LIN {X 0,Y 229.411,Z 367.195,A -85,B 0,C 180,E1 -21102.467,E2 -21102.467} C_VEL
LIN {X 0,Y 228.423,Z 377.715,A -85,B 0,C 180,E1 -21103.053,E2 -21103.053} C_VEL
LIN {X 0,Y 226.714,Z 389.278,A -85,B 0,C 180,E1 -21104.045,E2 -21104.045} C_VEL
LIN {X 0,Y 225.078,Z 397.764,A -85,B 0,C 180,E1 -21105.053,E2 -21105.053} C_VEL
LIN {X 0,Y 223.008,Z 406.34,A -85,B 0,C 180,E1 -21106.348,E2 -21106.348} C_VEL
LIN {X 0,Y 221.124,Z 413.107,A -85,B 0,C 180,E1 -21107.61,E2 -21107.61} C_VEL
LIN {X 0,Y 218.634,Z 420.799,A -85,B 0,C 180,E1 -21109.388,E2 -21109.388} C_VEL
LIN {X 0,Y 216.972,Z 425.412,A -85,B 0,C 180,E1 -21110.663,E2 -21110.663} C_VEL
LIN {X 0,Y 214.589,Z 431.432,A -85,B 0,C 180,E1 -21112.707,E2 -21112.707} C_VEL
LIN {X 0,Y 212.554,Z 436.048,A -85,B 0,C 180,E1 -21114.646,E2 -21114.646} C_VEL
LIN {X 0,Y 210.526,Z 440.403,A -85,B 0,C 180,E1 -21116.988,E2 -21116.988} C_VEL
LIN {X 0,Y 208.603,Z 444.082,A -85,B 0,C 180,E1 -21119.645,E2 -21119.645} C_VEL
LIN {X 0,Y 207.361,Z 446.196,A -85,B 0,C 180,E1 -21121.771,E2 -21121.771} C_VEL
LIN {X 0,Y 206.384,Z 447.588,A -85,B 0,C 180,E1 -21123.725,E2 -21123.725} C_VEL
LIN {X 0,Y 205.598,Z 448.503,A -85,B 0,C 180,E1 -21125.783,E2 -21125.783} C_VEL
LIN {X 0,Y 205.017,Z 448.806,A -85,B 0,C 180,E1 -21127.847,E2 -21127.847} C_VEL
LIN {X 0,Y 204.612,Z 448.539,A -85,B 0,C 180,E1 -21129.911,E2 -21129.911} C_VEL
LIN {X 0,Y 204.369,Z 447.762,A -85,B 0,C 180,E1 -21131.971,E2 -21131.971} C_VEL
LIN {X 0,Y 204.347,Z 446.209,A -85,B 0,C 180,E1 -21134.332,E2 -21134.332} C_VEL
LIN {X 0,Y 204.576,Z 443.416,A -85,B 0,C 180,E1 -21137.097,E2 -21137.097} C_VEL
LIN {X 0,Y 204.907,Z 440.635,A -85,B 0,C 180,E1 -21139.127,E2 -21139.127} C_VEL
LIN {X 0,Y 205.336,Z 437.209,A -85,B 0,C 180,E1 -21141.14,E2 -21141.14} C_VEL
LIN {X 0,Y 205.954,Z 432.897,A -85,B 0,C 180,E1 -21143.201,E2 -21143.201} C_VEL
LIN {X 0,Y 206.566,Z 428.044,A -85,B 0,C 180,E1 -21145.121,E2 -21145.121} C_VEL
LIN {X 0,Y 207.459,Z 421.98,A -85,B 0,C 180,E1 -21147.088,E2 -21147.088} C_VEL
LIN {X 0,Y 208.512,Z 414.595,A -85,B 0,C 180,E1 -21149.035,E2 -21149.035} C_VEL
LIN {X 0,Y 209.626,Z 406.687,A -85,B 0,C 180,E1 -21150.721,E2 -21150.721} C_VEL
LIN {X 0,Y 210.63,Z 398.846,A -85,B 0,C 180,E1 -21152.072,E2 -21152.072} C_VEL
LIN {X 0,Y 211.564,Z 389.853,A -85,B 0,C 180,E1 -21153.307,E2 -21153.307} C_VEL
LIN {X 0,Y 212.44,Z 379.124,A -85,B 0,C 180,E1 -21154.418,E2 -21154.418} C_VEL
LIN {X 0,Y 213.039,Z 367.681,A -85,B 0,C 180,E1 -21155.183,E2 -21155.183} C_VEL
LIN {X 0,Y 213.743,Z 344.69,A -85,B 0,C 180,E1 -21156.017,E2 -21156.017} C_VEL
LIN {X 0,Y 214.449,Z 316.245,A -85,B 0,C 180,E1 -21156.958,E2 -21156.958} C_VEL
LIN {X 0,Y 213.406,Z 311.932,A -85,B 0,C 180,E1 -21157.204,E2 -21157.204} C_VEL
LIN {X 0,Y 207.738,Z 296.649,A -85,B 0,C 180,E1 -21158.29,E2 -21158.29} C_VEL
LIN {X 0,Y 207.116,Z 294.495,A -85,B 0,C 180,E1 -21158.446,E2 -21158.446} C_VEL
LIN {X 0,Y 206.854,Z 294.531,A -85,B 0,C 180,E1 -21163.759,E2 -21163.759} C_VEL
LIN {X 0,Y 206.829,Z 294.533,A -85,B 0,C 180,E1 -21167.957,E2 -21167.957} C_VEL
LIN {X 0,Y 206.719,Z 294.549,A -85,B 0,C 180,E1 -21173.394,E2 -21173.394} C_VEL
LIN {X 0,Y 206.663,Z 294.553,A -85,B 0,C 180,E1 -21178.431,E2 -21178.431} C_VEL
LIN {X 0,Y 206.67,Z 294.546,A -85,B 0,C 180,E1 -21182.963,E2 -21182.963} C_VEL
LIN {X 0,Y 206.646,Z 294.553,A -85,B 0,C 180,E1 -21187.748,E2 -21187.748} C_VEL
LIN {X 0,Y 206.614,Z 294.561,A -85,B 0,C 180,E1 -21191.566,E2 -21191.566} C_VEL
LIN {X 0,Y 206.612,Z 294.559,A -85,B 0,C 180,E1 -21195.588,E2 -21195.588} C_VEL
LIN {X 0,Y 206.643,Z 294.555,A -85,B 0,C 180,E1 -21199.755,E2 -21199.755} C_VEL
LIN {X 0,Y 206.685,Z 294.55,A -85,B 0,C 180,E1 -21204.695,E2 -21204.695} C_VEL
LIN {X 0,Y 206.684,Z 294.549,A -85,B 0,C 180,E1 -21209.341,E2 -21209.341} C_VEL
LIN {X 0,Y 206.696,Z 294.55,A -85,B 0,C 180,E1 -21213.775,E2 -21213.775} C_VEL
LIN {X 0,Y 206.742,Z 294.526,A -85,B 0,C 180,E1 -21218.049,E2 -21218.049} C_VEL
LIN {X 0,Y 207.124,Z 294.503,A -85,B 0,C 180,E1 -21222.354,E2 -21222.354} C_VEL
LIN {X 0,Y 208.929,Z 312.159,A -85,B 0,C 180,E1 -21223.393,E2 -21223.393} C_VEL
LIN {X 0,Y 207.623,Z 366.937,A -85,B 0,C 180,E1 -21226.799,E2 -21226.799} C_VEL
LIN {X 0,Y 207.292,Z 379.206,A -85,B 0,C 180,E1 -21227.897,E2 -21227.897} C_VEL
LIN {X 0,Y 206.834,Z 390.233,A -85,B 0,C 180,E1 -21229.236,E2 -21229.236} C_VEL
LIN {X 0,Y 206.324,Z 400.757,A -85,B 0,C 180,E1 -21230.942,E2 -21230.942} C_VEL
LIN {X 0,Y 205.886,Z 409.682,A -85,B 0,C 180,E1 -21232.727,E2 -21232.727} C_VEL
LIN {X 0,Y 205.418,Z 419.232,A -85,B 0,C 180,E1 -21235.1,E2 -21235.1} C_VEL
LIN {X 0,Y 205.266,Z 425.662,A -85,B 0,C 180,E1 -21237.063,E2 -21237.063} C_VEL
LIN {X 0,Y 204.925,Z 432.222,A -85,B 0,C 180,E1 -21239.515,E2 -21239.515} C_VEL
LIN {X 0,Y 204.912,Z 437.509,A -85,B 0,C 180,E1 -21241.972,E2 -21241.972} C_VEL
LIN {X 0,Y 205.35,Z 442.572,A -85,B 0,C 180,E1 -21244.914,E2 -21244.914} C_VEL
LIN {X 0,Y 206.174,Z 446.28,A -85,B 0,C 180,E1 -21247.843,E2 -21247.843} C_VEL
LIN {X 0,Y 207.385,Z 448.706,A -85,B 0,C 180,E1 -21250.649,E2 -21250.649} C_VEL
LIN {X 0,Y 209.615,Z 450.18,A -85,B 0,C 180,E1 -21253.58,E2 -21253.58} C_VEL
LIN {X 0,Y 211.19,Z 450.591,A -85,B 0,C 180,E1 -21255.445,E2 -21255.445} C_VEL
LIN {X 0,Y 213.288,Z 450.479,A -85,B 0,C 180,E1 -21257.257,E2 -21257.257} C_VEL
LIN {X 0,Y 215.528,Z 449.821,A -85,B 0,C 180,E1 -21259.037,E2 -21259.037} C_VEL
LIN {X 0,Y 217.99,Z 448.714,A -85,B 0,C 180,E1 -21260.777,E2 -21260.777} C_VEL
LIN {X 0,Y 222.26,Z 446.105,A -85,B 0,C 180,E1 -21263.288,E2 -21263.288} C_VEL
LIN {X 0,Y 226.988,Z 442.34,A -85,B 0,C 180,E1 -21265.693,E2 -21265.693} C_VEL
LIN {X 0,Y 232.158,Z 437.117,A -85,B 0,C 180,E1 -21267.989,E2 -21267.989} C_VEL
LIN {X 0,Y 236.824,Z 431.622,A -85,B 0,C 180,E1 -21269.812,E2 -21269.812} C_VEL
LIN {X 0,Y 241.781,Z 424.82,A -85,B 0,C 180,E1 -21271.553,E2 -21271.553} C_VEL
LIN {X 0,Y 247.029,Z 416.545,A -85,B 0,C 180,E1 -21273.212,E2 -21273.212} C_VEL
LIN {X 0,Y 251.926,Z 407.174,A -85,B 0,C 180,E1 -21274.644,E2 -21274.644} C_VEL
LIN {X 0,Y 253.424,Z 404.07,A -85,B 0,C 180,E1 -21275.039,E2 -21275.039} C_VEL
LIN {X 0,Y 254.666,Z 401.027,A -85,B 0,C 180,E1 -21275.561,E2 -21275.561} C_VEL
LIN {X 0,Y 256.581,Z 392.474,A -85,B 0,C 180,E1 -21277.676,E2 -21277.676} C_VEL
LIN {X 0,Y 257.472,Z 389.198,A -85,B 0,C 180,E1 -21278.133,E2 -21278.133} C_VEL
LIN {X 0,Y 257.664,Z 388.604,A -85,B 0,C 180,E1 -21278.182,E2 -21278.182} C_VEL
LIN {X 0,Y 260.972,Z 377.957,A -85,B 0,C 180,E1 -21278.916,E2 -21278.916} C_VEL
LIN {X 0,Y 262.394,Z 372.569,A -85,B 0,C 180,E1 -21279.217,E2 -21279.217} C_VEL
LIN {X 0,Y 261.762,Z 370.849,A -85,B 0,C 180,E1 -21280.53,E2 -21280.53} C_VEL
LIN {X 0,Y 261.245,Z 369.295,A -85,B 0,C 180,E1 -21282.269,E2 -21282.269} C_VEL
LIN {X 0,Y 260.914,Z 369.054,A -85,B 0,C 180,E1 -21285.545,E2 -21285.545} C_VEL
LIN {X 0,Y 261.153,Z 369.578,A -85,B 0,C 180,E1 -21287,E2 -21287} C_VEL
LIN {X 0,Y 262.17,Z 372.974,A -85,B 0,C 180,E1 -21289.887,E2 -21289.887} C_VEL
LIN {X 0,Y 262.361,Z 373.577,A -85,B 0,C 180,E1 -21290.252,E2 -21290.252} C_VEL
LIN {X 0,Y 258.592,Z 387.877,A -85,B 0,C 180,E1 -21291.027,E2 -21291.027} C_VEL
LIN {X 0,Y 254.187,Z 400.181,A -85,B 0,C 180,E1 -21291.85,E2 -21291.85} C_VEL
LIN {X 0,Y 248.945,Z 411.733,A -85,B 0,C 180,E1 -21292.883,E2 -21292.883} C_VEL
LIN {X 0,Y 243.475,Z 421.754,A -85,B 0,C 180,E1 -21294.087,E2 -21294.087} C_VEL
LIN {X 0,Y 237.019,Z 431.728,A -85,B 0,C 180,E1 -21295.71,E2 -21295.71} C_VEL
LIN {X 0,Y 231.35,Z 439.3,A -85,B 0,C 180,E1 -21297.369,E2 -21297.369} C_VEL
LIN {X 0,Y 225.07,Z 446.659,A -85,B 0,C 180,E1 -21299.507,E2 -21299.507} C_VEL
LIN {X 0,Y 220.232,Z 451.53,A -85,B 0,C 180,E1 -21301.4,E2 -21301.4} C_VEL
LIN {X 0,Y 215.03,Z 456.023,A -85,B 0,C 180,E1 -21303.817,E2 -21303.817} C_VEL
LIN {X 0,Y 210.452,Z 459.369,A -85,B 0,C 180,E1 -21306.375,E2 -21306.375} C_VEL
LIN {X 0,Y 207.759,Z 461.023,A -85,B 0,C 180,E1 -21308.154,E2 -21308.154} C_VEL
LIN {X 0,Y 205.278,Z 462.198,A -85,B 0,C 180,E1 -21309.979,E2 -21309.979} C_VEL
LIN {X 0,Y 203.302,Z 462.83,A -85,B 0,C 180,E1 -21311.873,E2 -21311.873} C_VEL
LIN {X 0,Y 200.363,Z 462.941,A -85,B 0,C 180,E1 -21315.786,E2 -21315.786} C_VEL
LIN {X 0,Y 199.313,Z 462.261,A -85,B 0,C 180,E1 -21317.785,E2 -21317.785} C_VEL
LIN {X 0,Y 198.285,Z 459.599,A -85,B 0,C 180,E1 -21321.849,E2 -21321.849} C_VEL
LIN {X 0,Y 198.2,Z 458.32,A -85,B 0,C 180,E1 -21323.293,E2 -21323.293} C_VEL
LIN {X 0,Y 197.665,Z 461.871,A -85,B 0,C 180,E1 -21325.922,E2 -21325.922} C_VEL
LIN {X 0,Y 197.59,Z 463.98,A -85,B 0,C 180,E1 -21327.961,E2 -21327.961} C_VEL
LIN {X 0,Y 197.617,Z 465.545,A -85,B 0,C 180,E1 -21330,E2 -21330} C_VEL
LIN {X 0,Y 197.498,Z 466.482,A -85,B 0,C 180,E1 -21332.039,E2 -21332.039} C_VEL
LIN {X 0,Y 197.419,Z 466.975,A -85,B 0,C 180,E1 -21334.542,E2 -21334.542} C_VEL
LIN {X 0,Y 197.725,Z 466.437,A -85,B 0,C 180,E1 -21338.173,E2 -21338.173} C_VEL
LIN {X 0,Y 198.227,Z 465.424,A -85,B 0,C 180,E1 -21340.21,E2 -21340.21} C_VEL
LIN {X 0,Y 199.459,Z 462.979,A -85,B 0,C 180,E1 -21343.24,E2 -21343.24} C_VEL
LIN {X 0,Y 201.207,Z 459.238,A -85,B 0,C 180,E1 -21346.226,E2 -21346.226} C_VEL
LIN {X 0,Y 202.731,Z 456.069,A -85,B 0,C 180,E1 -21348.179,E2 -21348.179} C_VEL
LIN {X 0,Y 205.071,Z 451.053,A -85,B 0,C 180,E1 -21350.565,E2 -21350.565} C_VEL
LIN {X 0,Y 207.767,Z 444.774,A -85,B 0,C 180,E1 -21352.892,E2 -21352.892} C_VEL
LIN {X 0,Y 210.188,Z 438.652,A -85,B 0,C 180,E1 -21354.705,E2 -21354.705} C_VEL
LIN {X 0,Y 212.071,Z 433.271,A -85,B 0,C 180,E1 -21356.046,E2 -21356.046} C_VEL
LIN {X 0,Y 214.178,Z 426.968,A -85,B 0,C 180,E1 -21357.348,E2 -21357.348} C_VEL
LIN {X 0,Y 216.962,Z 417.427,A -85,B 0,C 180,E1 -21358.886,E2 -21358.886} C_VEL
LIN {X 0,Y 218.812,Z 409.826,A -85,B 0,C 180,E1 -21359.856,E2 -21359.856} C_VEL
LIN {X 0,Y 220.554,Z 401.702,A -85,B 0,C 180,E1 -21360.653,E2 -21360.653} C_VEL
LIN {X 0,Y 222.104,Z 392.178,A -85,B 0,C 180,E1 -21361.346,E2 -21361.346} C_VEL
LIN {X 0,Y 223.067,Z 382.979,A -85,B 0,C 180,E1 -21361.814,E2 -21361.814} C_VEL
LIN {X 0,Y 224.088,Z 362.598,A -85,B 0,C 180,E1 -21362.502,E2 -21362.502} C_VEL
LIN {X 0,Y 221.37,Z 343.446,A -85,B 0,C 180,E1 -21363.879,E2 -21363.879} C_VEL
LIN {X 0,Y 220.472,Z 339.745,A -85,B 0,C 180,E1 -21364.235,E2 -21364.235} C_VEL
LIN {X 0,Y 215.073,Z 327.747,A -85,B 0,C 180,E1 -21366.016,E2 -21366.016} C_VEL
LIN {X 0,Y 209.948,Z 317.918,A -85,B 0,C 180,E1 -21367.766,E2 -21367.766} C_VEL
LIN {X 0,Y 207.328,Z 313.245,A -85,B 0,C 180,E1 -21368.696,E2 -21368.696} C_VEL
LIN {X 0,Y 204.763,Z 308.846,A -85,B 0,C 180,E1 -21369.638,E2 -21369.638} C_VEL
LIN {X 0,Y 202.164,Z 304.496,A -85,B 0,C 180,E1 -21370.632,E2 -21370.632} C_VEL
LIN {X 0,Y 201.935,Z 303.874,A -85,B 0,C 180,E1 -21370.819,E2 -21370.819} C_VEL
LIN {X 0,Y 200.406,Z 298.59,A -85,B 0,C 180,E1 -21374.537,E2 -21374.537} C_VEL
LIN {X 0,Y 199.607,Z 295.427,A -85,B 0,C 180,E1 -21377.05,E2 -21377.05} C_VEL
LIN {X 0,Y 199.606,Z 295.424,A -85,B 0,C 180,E1 -21380.769,E2 -21380.769} C_VEL
LIN {X 0,Y 199.619,Z 295.423,A -85,B 0,C 180,E1 -21385.708,E2 -21385.708} C_VEL
LIN {X 0,Y 199.694,Z 295.414,A -85,B 0,C 180,E1 -21388.13,E2 -21388.13} C_VEL
LIN {X 0,Y 199.651,Z 295.419,A -85,B 0,C 180,E1 -21392.76,E2 -21392.76} C_VEL
LIN {X 0,Y 199.715,Z 295.413,A -85,B 0,C 180,E1 -21397.22,E2 -21397.22} C_VEL
LIN {X 0,Y 199.801,Z 295.405,A -85,B 0,C 180,E1 -21401.754,E2 -21401.754} C_VEL
LIN {X 0,Y 199.828,Z 295.4,A -85,B 0,C 180,E1 -21405.742,E2 -21405.742} C_VEL
LIN {X 0,Y 200.026,Z 295.362,A -85,B 0,C 180,E1 -21409.876,E2 -21409.876} C_VEL
LIN {X 0,Y 200.02,Z 295.362,A -85,B 0,C 180,E1 -21413.943,E2 -21413.943} C_VEL
LIN {X 0,Y 200.316,Z 295.336,A -85,B 0,C 180,E1 -21417.983,E2 -21417.983} C_VEL
LIN {X 0,Y 200.473,Z 295.305,A -85,B 0,C 180,E1 -21419.994,E2 -21419.994} C_VEL
LIN {X 0,Y 200.016,Z 295.37,A -85,B 0,C 180,E1 -21424.023,E2 -21424.023} C_VEL
LIN {X 0,Y 200.079,Z 295.374,A -85,B 0,C 180,E1 -21428.07,E2 -21428.07} C_VEL
LIN {X 0,Y 199.87,Z 295.395,A -85,B 0,C 180,E1 -21432.173,E2 -21432.173} C_VEL
LIN {X 0,Y 199.797,Z 295.398,A -85,B 0,C 180,E1 -21436.337,E2 -21436.337} C_VEL
LIN {X 0,Y 199.694,Z 295.411,A -85,B 0,C 180,E1 -21440.598,E2 -21440.598} C_VEL
LIN {X 0,Y 199.662,Z 295.418,A -85,B 0,C 180,E1 -21444.978,E2 -21444.978} C_VEL
LIN {X 0,Y 199.651,Z 295.425,A -85,B 0,C 180,E1 -21449.517,E2 -21449.517} C_VEL
LIN {X 0,Y 199.677,Z 295.469,A -85,B 0,C 180,E1 -21451.784,E2 -21451.784} C_VEL
LIN {X 0,Y 200.481,Z 297.963,A -85,B 0,C 180,E1 -21452.178,E2 -21452.178} C_VEL
LIN {X 0,Y 202.382,Z 300.199,A -85,B 0,C 180,E1 -21452.885,E2 -21452.885} C_VEL
LIN {X 0,Y 203.114,Z 301.083,A -85,B 0,C 180,E1 -21453.153,E2 -21453.153} C_VEL
LIN {X 0,Y 205.286,Z 304.358,A -85,B 0,C 180,E1 -21453.958,E2 -21453.958} C_VEL
LIN {X 0,Y 210.304,Z 311.674,A -85,B 0,C 180,E1 -21455.703,E2 -21455.703} C_VEL
LIN {X 0,Y 216.59,Z 321.533,A -85,B 0,C 180,E1 -21457.743,E2 -21457.743} C_VEL
LIN {X 0,Y 222.99,Z 333.019,A -85,B 0,C 180,E1 -21459.703,E2 -21459.703} C_VEL
LIN {X 0,Y 225.333,Z 338.511,A -85,B 0,C 180,E1 -21460.432,E2 -21460.432} C_VEL
LIN {X 0,Y 223.827,Z 366.884,A -85,B 0,C 180,E1 -21461.355,E2 -21461.355} C_VEL
LIN {X 0,Y 222.95,Z 376.004,A -85,B 0,C 180,E1 -21461.841,E2 -21461.841} C_VEL
LIN {X 0,Y 221.602,Z 385.861,A -85,B 0,C 180,E1 -21462.623,E2 -21462.623} C_VEL
LIN {X 0,Y 219.46,Z 397.28,A -85,B 0,C 180,E1 -21463.901,E2 -21463.901} C_VEL
LIN {X 0,Y 217.173,Z 406.269,A -85,B 0,C 180,E1 -21465.259,E2 -21465.259} C_VEL
LIN {X 0,Y 214.687,Z 414.699,A -85,B 0,C 180,E1 -21466.893,E2 -21466.893} C_VEL
LIN {X 0,Y 212.346,Z 421.559,A -85,B 0,C 180,E1 -21468.552,E2 -21468.552} C_VEL
LIN {X 0,Y 209.84,Z 428.001,A -85,B 0,C 180,E1 -21470.48,E2 -21470.48} C_VEL
LIN {X 0,Y 206.985,Z 434.507,A -85,B 0,C 180,E1 -21472.938,E2 -21472.938} C_VEL
LIN {X 0,Y 204.46,Z 439.725,A -85,B 0,C 180,E1 -21475.571,E2 -21475.571} C_VEL
LIN {X 0,Y 202.141,Z 443.96,A -85,B 0,C 180,E1 -21478.566,E2 -21478.566} C_VEL
LIN {X 0,Y 200.544,Z 446.53,A -85,B 0,C 180,E1 -21481.16,E2 -21481.16} C_VEL
LIN {X 0,Y 199.69,Z 447.732,A -85,B 0,C 180,E1 -21482.773,E2 -21482.773} C_VEL
LIN {X 0,Y 198.808,Z 448.703,A -85,B 0,C 180,E1 -21484.9,E2 -21484.9} C_VEL
LIN {X 0,Y 198.061,Z 449.116,A -85,B 0,C 180,E1 -21487.285,E2 -21487.285} C_VEL
LIN {X 0,Y 197.642,Z 448.943,A -85,B 0,C 180,E1 -21489.171,E2 -21489.171} C_VEL
LIN {X 0,Y 197.328,Z 448.293,A -85,B 0,C 180,E1 -21491.305,E2 -21491.305} C_VEL
LIN {X 0,Y 197.254,Z 446.572,A -85,B 0,C 180,E1 -21494.12,E2 -21494.12} C_VEL
LIN {X 0,Y 197.411,Z 444.21,A -85,B 0,C 180,E1 -21496.621,E2 -21496.621} C_VEL
LIN {X 0,Y 197.924,Z 439.995,A -85,B 0,C 180,E1 -21499.774,E2 -21499.774} C_VEL
LIN {X 0,Y 198.554,Z 435.513,A -85,B 0,C 180,E1 -21502.28,E2 -21502.28} C_VEL
LIN {X 0,Y 199.396,Z 429.454,A -85,B 0,C 180,E1 -21504.945,E2 -21504.945} C_VEL
LIN {X 0,Y 200.517,Z 421.898,A -85,B 0,C 180,E1 -21507.489,E2 -21507.489} C_VEL
LIN {X 0,Y 201.603,Z 414.437,A -85,B 0,C 180,E1 -21509.501,E2 -21509.501} C_VEL
LIN {X 0,Y 202.77,Z 406.431,A -85,B 0,C 180,E1 -21511.242,E2 -21511.242} C_VEL
LIN {X 0,Y 204.042,Z 396.843,A -85,B 0,C 180,E1 -21512.894,E2 -21512.894} C_VEL
LIN {X 0,Y 205.137,Z 385.908,A -85,B 0,C 180,E1 -21514.298,E2 -21514.298} C_VEL
LIN {X 0,Y 205.853,Z 376.021,A -85,B 0,C 180,E1 -21515.204,E2 -21515.204} C_VEL
LIN {X 0,Y 206.3,Z 366.415,A -85,B 0,C 180,E1 -21515.805,E2 -21515.805} C_VEL
LIN {X 0,Y 207.728,Z 317.216,A -85,B 0,C 180,E1 -21517.537,E2 -21517.537} C_VEL
LIN {X 0,Y 206.282,Z 312.34,A -85,B 0,C 180,E1 -21517.854,E2 -21517.854} C_VEL
LIN {X 0,Y 200.994,Z 298.072,A -85,B 0,C 180,E1 -21518.919,E2 -21518.919} C_VEL
LIN {X 0,Y 200.042,Z 295.378,A -85,B 0,C 180,E1 -21519.162,E2 -21519.162} C_VEL
LIN {X 0,Y 199.795,Z 295.41,A -85,B 0,C 180,E1 -21524.255,E2 -21524.255} C_VEL
LIN {X 0,Y 199.754,Z 295.414,A -85,B 0,C 180,E1 -21528.461,E2 -21528.461} C_VEL
LIN {X 0,Y 199.681,Z 295.426,A -85,B 0,C 180,E1 -21533.801,E2 -21533.801} C_VEL
LIN {X 0,Y 199.64,Z 295.428,A -85,B 0,C 180,E1 -21538.365,E2 -21538.365} C_VEL
LIN {X 0,Y 199.641,Z 295.42,A -85,B 0,C 180,E1 -21542.357,E2 -21542.357} C_VEL
LIN {X 0,Y 199.595,Z 295.432,A -85,B 0,C 180,E1 -21546.77,E2 -21546.77} C_VEL
LIN {X 0,Y 199.574,Z 295.433,A -85,B 0,C 180,E1 -21549.337,E2 -21549.337} C_VEL
LIN {X 0,Y 199.548,Z 295.438,A -85,B 0,C 180,E1 -21552.314,E2 -21552.314} C_VEL
LIN {X 0,Y 199.558,Z 295.436,A -85,B 0,C 180,E1 -21555.234,E2 -21555.234} C_VEL
LIN {X 0,Y 199.561,Z 295.439,A -85,B 0,C 180,E1 -21558.011,E2 -21558.011} C_VEL
LIN {X 0,Y 199.594,Z 295.429,A -85,B 0,C 180,E1 -21560.774,E2 -21560.774} C_VEL
LIN {X 0,Y 199.598,Z 295.435,A -85,B 0,C 180,E1 -21565.72,E2 -21565.72} C_VEL
LIN {X 0,Y 199.673,Z 295.422,A -85,B 0,C 180,E1 -21568.141,E2 -21568.141} C_VEL
LIN {X 0,Y 199.633,Z 295.428,A -85,B 0,C 180,E1 -21572.772,E2 -21572.772} C_VEL
LIN {X 0,Y 199.706,Z 295.407,A -85,B 0,C 180,E1 -21577.233,E2 -21577.233} C_VEL
LIN {X 0,Y 200.111,Z 295.348,A -85,B 0,C 180,E1 -21582.474,E2 -21582.474} C_VEL
LIN {X 0,Y 201.834,Z 312.319,A -85,B 0,C 180,E1 -21583.508,E2 -21583.508} C_VEL
LIN {X 0,Y 200.597,Z 367.18,A -85,B 0,C 180,E1 -21587.101,E2 -21587.101} C_VEL
LIN {X 0,Y 200.255,Z 379.24,A -85,B 0,C 180,E1 -21588.237,E2 -21588.237} C_VEL
LIN {X 0,Y 199.831,Z 390.259,A -85,B 0,C 180,E1 -21589.623,E2 -21589.623} C_VEL
LIN {X 0,Y 199.322,Z 400.561,A -85,B 0,C 180,E1 -21591.337,E2 -21591.337} C_VEL
LIN {X 0,Y 198.883,Z 409.612,A -85,B 0,C 180,E1 -21593.196,E2 -21593.196} C_VEL
LIN {X 0,Y 198.46,Z 418.538,A -85,B 0,C 180,E1 -21595.437,E2 -21595.437} C_VEL
LIN {X 0,Y 198.182,Z 426.454,A -85,B 0,C 180,E1 -21597.974,E2 -21597.974} C_VEL
LIN {X 0,Y 197.944,Z 432.845,A -85,B 0,C 180,E1 -21600.515,E2 -21600.515} C_VEL
LIN {X 0,Y 198.036,Z 438.096,A -85,B 0,C 180,E1 -21603.058,E2 -21603.058} C_VEL
LIN {X 0,Y 198.602,Z 443.122,A -85,B 0,C 180,E1 -21606.1,E2 -21606.1} C_VEL
LIN {X 0,Y 199.488,Z 446.591,A -85,B 0,C 180,E1 -21608.97,E2 -21608.97} C_VEL
LIN {X 0,Y 201.08,Z 449.222,A -85,B 0,C 180,E1 -21612.111,E2 -21612.111} C_VEL
LIN {X 0,Y 202.736,Z 450.356,A -85,B 0,C 180,E1 -21614.05,E2 -21614.05} C_VEL
LIN {X 0,Y 204.366,Z 450.922,A -85,B 0,C 180,E1 -21615.975,E2 -21615.975} C_VEL
LIN {X 0,Y 206.556,Z 451.016,A -85,B 0,C 180,E1 -21617.838,E2 -21617.838} C_VEL
LIN {X 0,Y 210.298,Z 450.288,A -85,B 0,C 180,E1 -21620.651,E2 -21620.651} C_VEL
LIN {X 0,Y 214.348,Z 448.578,A -85,B 0,C 180,E1 -21623.175,E2 -21623.175} C_VEL
LIN {X 0,Y 219.13,Z 445.649,A -85,B 0,C 180,E1 -21625.662,E2 -21625.662} C_VEL
LIN {X 0,Y 224.371,Z 441.435,A -85,B 0,C 180,E1 -21628.03,E2 -21628.03} C_VEL
LIN {X 0,Y 230.072,Z 435.822,A -85,B 0,C 180,E1 -21630.272,E2 -21630.272} C_VEL
LIN {X 0,Y 236.198,Z 428.724,A -85,B 0,C 180,E1 -21632.389,E2 -21632.389} C_VEL
LIN {X 0,Y 241.606,Z 421.119,A -85,B 0,C 180,E1 -21634.058,E2 -21634.058} C_VEL
LIN {X 0,Y 247.87,Z 410.793,A -85,B 0,C 180,E1 -21635.793,E2 -21635.793} C_VEL
LIN {X 0,Y 252.598,Z 401.229,A -85,B 0,C 180,E1 -21636.994,E2 -21636.994} C_VEL
LIN {X 0,Y 256.461,Z 391.834,A -85,B 0,C 180,E1 -21637.913,E2 -21637.913} C_VEL
LIN {X 0,Y 257.664,Z 388.604,A -85,B 0,C 180,E1 -21638.182,E2 -21638.182} C_VEL
LIN {X 0,Y 258.662,Z 385.151,A -85,B 0,C 180,E1 -21638.594,E2 -21638.594} C_VEL
LIN {X 0,Y 259.267,Z 382.229,A -85,B 0,C 180,E1 -21639.215,E2 -21639.215} C_VEL
LIN {X 0,Y 259.504,Z 379.196,A -85,B 0,C 180,E1 -21640.245,E2 -21640.245} C_VEL
LIN {X 0,Y 259.415,Z 377.14,A -85,B 0,C 180,E1 -21641.413,E2 -21641.413} C_VEL
LIN {X 0,Y 259.3,Z 376.514,A -85,B 0,C 180,E1 -21642.025,E2 -21642.025} C_VEL
LIN {X 0,Y 259.142,Z 375.939,A -85,B 0,C 180,E1 -21642.924,E2 -21642.924} C_VEL
LIN {X 0,Y 259.164,Z 376.017,A -85,B 0,C 180,E1 -21646.177,E2 -21646.177} C_VEL
LIN {X 0,Y 259.289,Z 376.947,A -85,B 0,C 180,E1 -21647.341,E2 -21647.341} C_VEL
LIN {X 0,Y 259.732,Z 378.763,A -85,B 0,C 180,E1 -21648.975,E2 -21648.975} C_VEL
LIN {X 0,Y 255.364,Z 392.759,A -85,B 0,C 180,E1 -21649.758,E2 -21649.758} C_VEL
LIN {X 0,Y 250.507,Z 404.326,A -85,B 0,C 180,E1 -21650.598,E2 -21650.598} C_VEL
LIN {X 0,Y 245.588,Z 413.986,A -85,B 0,C 180,E1 -21651.506,E2 -21651.506} C_VEL
LIN {X 0,Y 238.777,Z 425.141,A -85,B 0,C 180,E1 -21652.94,E2 -21652.94} C_VEL
LIN {X 0,Y 232.723,Z 433.557,A -85,B 0,C 180,E1 -21654.402,E2 -21654.402} C_VEL
LIN {X 0,Y 225.565,Z 442.07,A -85,B 0,C 180,E1 -21656.424,E2 -21656.424} C_VEL
LIN {X 0,Y 220.142,Z 447.633,A -85,B 0,C 180,E1 -21658.213,E2 -21658.213} C_VEL
LIN {X 0,Y 214.115,Z 452.944,A -85,B 0,C 180,E1 -21660.504,E2 -21660.504} C_VEL
LIN {X 0,Y 208.732,Z 457.02,A -85,B 0,C 180,E1 -21662.964,E2 -21662.964} C_VEL
LIN {X 0,Y 203.987,Z 459.927,A -85,B 0,C 180,E1 -21665.578,E2 -21665.578} C_VEL
LIN {X 0,Y 201.199,Z 461.212,A -85,B 0,C 180,E1 -21667.403,E2 -21667.403} C_VEL
LIN {X 0,Y 198.633,Z 462.088,A -85,B 0,C 180,E1 -21669.278,E2 -21669.278} C_VEL
LIN {X 0,Y 196.563,Z 462.583,A -85,B 0,C 180,E1 -21671.228,E2 -21671.228} C_VEL
LIN {X 0,Y 194.886,Z 462.545,A -85,B 0,C 180,E1 -21673.232,E2 -21673.232} C_VEL
LIN {X 0,Y 192.448,Z 461.243,A -85,B 0,C 180,E1 -21677.343,E2 -21677.343} C_VEL
LIN {X 0,Y 191.732,Z 459.964,A -85,B 0,C 180,E1 -21679.439,E2 -21679.439} C_VEL
LIN {X 0,Y 191.314,Z 457.197,A -85,B 0,C 180,E1 -21682.719,E2 -21682.719} C_VEL
LIN {X 0,Y 190.586,Z 461.295,A -85,B 0,C 180,E1 -21685.77,E2 -21685.77} C_VEL
LIN {X 0,Y 190.511,Z 463.478,A -85,B 0,C 180,E1 -21687.885,E2 -21687.885} C_VEL
LIN {X 0,Y 190.552,Z 465.071,A -85,B 0,C 180,E1 -21690,E2 -21690} C_VEL
LIN {X 0,Y 190.413,Z 466.049,A -85,B 0,C 180,E1 -21692.115,E2 -21692.115} C_VEL
LIN {X 0,Y 190.345,Z 466.58,A -85,B 0,C 180,E1 -21694.449,E2 -21694.449} C_VEL
LIN {X 0,Y 190.394,Z 466.605,A -85,B 0,C 180,E1 -21696.357,E2 -21696.357} C_VEL
LIN {X 0,Y 190.7,Z 466.194,A -85,B 0,C 180,E1 -21698.477,E2 -21698.477} C_VEL
LIN {X 0,Y 191.245,Z 465.199,A -85,B 0,C 180,E1 -21700.587,E2 -21700.587} C_VEL
LIN {X 0,Y 192.045,Z 463.712,A -85,B 0,C 180,E1 -21702.684,E2 -21702.684} C_VEL
LIN {X 0,Y 193.727,Z 460.567,A -85,B 0,C 180,E1 -21705.788,E2 -21705.788} C_VEL
LIN {X 0,Y 196.008,Z 456.134,A -85,B 0,C 180,E1 -21708.826,E2 -21708.826} C_VEL
LIN {X 0,Y 198.951,Z 450.055,A -85,B 0,C 180,E1 -21711.772,E2 -21711.772} C_VEL
LIN {X 0,Y 201.263,Z 445.057,A -85,B 0,C 180,E1 -21713.676,E2 -21713.676} C_VEL
LIN {X 0,Y 203.788,Z 439.064,A -85,B 0,C 180,E1 -21715.536,E2 -21715.536} C_VEL
LIN {X 0,Y 206.125,Z 432.82,A -85,B 0,C 180,E1 -21717.131,E2 -21717.131} C_VEL
LIN {X 0,Y 208.435,Z 426.133,A -85,B 0,C 180,E1 -21718.525,E2 -21718.525} C_VEL
LIN {X 0,Y 211.082,Z 417.402,A -85,B 0,C 180,E1 -21719.962,E2 -21719.962} C_VEL
LIN {X 0,Y 213.259,Z 408.849,A -85,B 0,C 180,E1 -21721.061,E2 -21721.061} C_VEL
LIN {X 0,Y 215.246,Z 399.843,A -85,B 0,C 180,E1 -21721.918,E2 -21721.918} C_VEL
LIN {X 0,Y 216.809,Z 389.95,A -85,B 0,C 180,E1 -21722.613,E2 -21722.613} C_VEL
LIN {X 0,Y 217.827,Z 378.916,A -85,B 0,C 180,E1 -21723.13,E2 -21723.13} C_VEL
LIN {X 0,Y 218.53,Z 363.247,A -85,B 0,C 180,E1 -21723.653,E2 -21723.653} C_VEL
LIN {X 0,Y 216.028,Z 345.32,A -85,B 0,C 180,E1 -21725.001,E2 -21725.001} C_VEL
LIN {X 0,Y 215.131,Z 342.296,A -85,B 0,C 180,E1 -21725.346,E2 -21725.346} C_VEL
LIN {X 0,Y 210.16,Z 331.327,A -85,B 0,C 180,E1 -21727.076,E2 -21727.076} C_VEL
LIN {X 0,Y 205.162,Z 321.484,A -85,B 0,C 180,E1 -21728.897,E2 -21728.897} C_VEL
LIN {X 0,Y 200.74,Z 313.714,A -85,B 0,C 180,E1 -21730.583,E2 -21730.583} C_VEL
LIN {X 0,Y 197.579,Z 308.57,A -85,B 0,C 180,E1 -21731.854,E2 -21731.854} C_VEL
LIN {X 0,Y 195.033,Z 304.482,A -85,B 0,C 180,E1 -21732.943,E2 -21732.943} C_VEL
LIN {X 0,Y 194.587,Z 303.445,A -85,B 0,C 180,E1 -21733.189,E2 -21733.189} C_VEL
LIN {X 0,Y 192.521,Z 296.365,A -85,B 0,C 180,E1 -21738.764,E2 -21738.764} C_VEL
LIN {X 0,Y 192.591,Z 296.304,A -85,B 0,C 180,E1 -21743.4,E2 -21743.4} C_VEL
LIN {X 0,Y 192.614,Z 296.305,A -85,B 0,C 180,E1 -21747.056,E2 -21747.056} C_VEL
LIN {X 0,Y 192.643,Z 296.3,A -85,B 0,C 180,E1 -21751.682,E2 -21751.682} C_VEL
LIN {X 0,Y 192.686,Z 296.296,A -85,B 0,C 180,E1 -21756.34,E2 -21756.34} C_VEL
LIN {X 0,Y 192.736,Z 296.288,A -85,B 0,C 180,E1 -21761.454,E2 -21761.454} C_VEL
LIN {X 0,Y 192.757,Z 296.276,A -85,B 0,C 180,E1 -21765.207,E2 -21765.207} C_VEL
LIN {X 0,Y 192.949,Z 296.242,A -85,B 0,C 180,E1 -21769.56,E2 -21769.56} C_VEL
LIN {X 0,Y 193.04,Z 296.246,A -85,B 0,C 180,E1 -21771.62,E2 -21771.62} C_VEL
LIN {X 0,Y 193.258,Z 296.216,A -85,B 0,C 180,E1 -21777.909,E2 -21777.909} C_VEL
LIN {X 0,Y 193.437,Z 296.181,A -85,B 0,C 180,E1 -21779.993,E2 -21779.993} C_VEL
LIN {X 0,Y 192.961,Z 296.247,A -85,B 0,C 180,E1 -21784.17,E2 -21784.17} C_VEL
LIN {X 0,Y 193.028,Z 296.251,A -85,B 0,C 180,E1 -21788.367,E2 -21788.367} C_VEL
LIN {X 0,Y 192.797,Z 296.279,A -85,B 0,C 180,E1 -21792.626,E2 -21792.626} C_VEL
LIN {X 0,Y 192.75,Z 296.279,A -85,B 0,C 180,E1 -21796.952,E2 -21796.952} C_VEL
LIN {X 0,Y 192.63,Z 296.294,A -85,B 0,C 180,E1 -21801.39,E2 -21801.39} C_VEL
LIN {X 0,Y 192.654,Z 296.29,A -85,B 0,C 180,E1 -21804.218,E2 -21804.218} C_VEL
LIN {X 0,Y 192.643,Z 296.463,A -85,B 0,C 180,E1 -21809.409,E2 -21809.409} C_VEL
LIN {X 0,Y 193.582,Z 299.117,A -85,B 0,C 180,E1 -21809.906,E2 -21809.906} C_VEL
LIN {X 0,Y 195.69,Z 301.304,A -85,B 0,C 180,E1 -21810.773,E2 -21810.773} C_VEL
LIN {X 0,Y 196.798,Z 303.108,A -85,B 0,C 180,E1 -21811.252,E2 -21811.252} C_VEL
LIN {X 0,Y 199.092,Z 306.03,A -85,B 0,C 180,E1 -21812.168,E2 -21812.168} C_VEL
LIN {X 0,Y 207.882,Z 318.968,A -85,B 0,C 180,E1 -21815.405,E2 -21815.405} C_VEL
LIN {X 0,Y 215.07,Z 331.068,A -85,B 0,C 180,E1 -21817.807,E2 -21817.807} C_VEL
LIN {X 0,Y 218.953,Z 338.651,A -85,B 0,C 180,E1 -21819.049,E2 -21819.049} C_VEL
LIN {X 0,Y 219.761,Z 340.586,A -85,B 0,C 180,E1 -21819.315,E2 -21819.315} C_VEL
LIN {X 0,Y 218.221,Z 368.422,A -85,B 0,C 180,E1 -21820.258,E2 -21820.258} C_VEL
LIN {X 0,Y 217.141,Z 378.818,A -85,B 0,C 180,E1 -21820.87,E2 -21820.87} C_VEL
LIN {X 0,Y 215.498,Z 388.985,A -85,B 0,C 180,E1 -21821.754,E2 -21821.754} C_VEL
LIN {X 0,Y 213.505,Z 398.457,A -85,B 0,C 180,E1 -21822.912,E2 -21822.912} C_VEL
LIN {X 0,Y 211.318,Z 406.613,A -85,B 0,C 180,E1 -21824.172,E2 -21824.172} C_VEL
LIN {X 0,Y 208.909,Z 414.517,A -85,B 0,C 180,E1 -21825.729,E2 -21825.729} C_VEL
LIN {X 0,Y 206.791,Z 420.563,A -85,B 0,C 180,E1 -21827.179,E2 -21827.179} C_VEL
LIN {X 0,Y 204.1,Z 427.219,A -85,B 0,C 180,E1 -21829.138,E2 -21829.138} C_VEL
LIN {X 0,Y 201.626,Z 432.686,A -85,B 0,C 180,E1 -21831.14,E2 -21831.14} C_VEL
LIN {X 0,Y 199.41,Z 437.189,A -85,B 0,C 180,E1 -21833.192,E2 -21833.192} C_VEL
LIN {X 0,Y 197.46,Z 440.873,A -85,B 0,C 180,E1 -21835.287,E2 -21835.287} C_VEL
LIN {X 0,Y 195.011,Z 445.028,A -85,B 0,C 180,E1 -21838.496,E2 -21838.496} C_VEL
LIN {X 0,Y 193.074,Z 447.81,A -85,B 0,C 180,E1 -21841.758,E2 -21841.758} C_VEL
LIN {X 0,Y 192.053,Z 448.851,A -85,B 0,C 180,E1 -21843.952,E2 -21843.952} C_VEL
LIN {X 0,Y 191.065,Z 449.449,A -85,B 0,C 180,E1 -21846.843,E2 -21846.843} C_VEL
LIN {X 0,Y 190.32,Z 448.822,A -85,B 0,C 180,E1 -21850.589,E2 -21850.589} C_VEL
LIN {X 0,Y 190.166,Z 446.934,A -85,B 0,C 180,E1 -21853.89,E2 -21853.89} C_VEL
LIN {X 0,Y 190.379,Z 443.792,A -85,B 0,C 180,E1 -21857.204,E2 -21857.204} C_VEL
LIN {X 0,Y 190.978,Z 439.328,A -85,B 0,C 180,E1 -21860.468,E2 -21860.468} C_VEL
LIN {X 0,Y 191.707,Z 434.304,A -85,B 0,C 180,E1 -21863.17,E2 -21863.17} C_VEL
LIN {X 0,Y 192.574,Z 428.009,A -85,B 0,C 180,E1 -21865.815,E2 -21865.815} C_VEL
LIN {X 0,Y 193.564,Z 421.805,A -85,B 0,C 180,E1 -21867.92,E2 -21867.92} C_VEL
LIN {X 0,Y 194.551,Z 415.3,A -85,B 0,C 180,E1 -21869.742,E2 -21869.742} C_VEL
LIN {X 0,Y 195.75,Z 407.402,A -85,B 0,C 180,E1 -21871.543,E2 -21871.543} C_VEL
LIN {X 0,Y 196.93,Z 398.94,A -85,B 0,C 180,E1 -21873.089,E2 -21873.089} C_VEL
LIN {X 0,Y 198.097,Z 388.482,A -85,B 0,C 180,E1 -21874.579,E2 -21874.579} C_VEL
LIN {X 0,Y 198.97,Z 377.252,A -85,B 0,C 180,E1 -21875.702,E2 -21875.702} C_VEL
LIN {X 0,Y 199.503,Z 367.398,A -85,B 0,C 180,E1 -21876.355,E2 -21876.355} C_VEL
LIN {X 0,Y 200.598,Z 333.822,A -85,B 0,C 180,E1 -21877.598,E2 -21877.598} C_VEL
LIN {X 0,Y 200.939,Z 317.741,A -85,B 0,C 180,E1 -21878.175,E2 -21878.175} C_VEL
LIN {X 0,Y 195.014,Z 301.589,A -85,B 0,C 180,E1 -21879.42,E2 -21879.42} C_VEL
LIN {X 0,Y 193.128,Z 297.058,A -85,B 0,C 180,E1 -21879.809,E2 -21879.809} C_VEL
LIN {X 0,Y 192.998,Z 296.259,A -85,B 0,C 180,E1 -21879.86,E2 -21879.86} C_VEL
LIN {X 0,Y 192.725,Z 296.292,A -85,B 0,C 180,E1 -21884.79,E2 -21884.79} C_VEL
LIN {X 0,Y 192.66,Z 296.3,A -85,B 0,C 180,E1 -21889.167,E2 -21889.167} C_VEL
LIN {X 0,Y 192.613,Z 296.305,A -85,B 0,C 180,E1 -21894.211,E2 -21894.211} C_VEL
LIN {X 0,Y 192.576,Z 296.308,A -85,B 0,C 180,E1 -21898.87,E2 -21898.87} C_VEL
LIN {X 0,Y 192.571,Z 296.302,A -85,B 0,C 180,E1 -21903.192,E2 -21903.192} C_VEL
LIN {X 0,Y 192.52,Z 296.31,A -85,B 0,C 180,E1 -21908.36,E2 -21908.36} C_VEL
LIN {X 0,Y 192.467,Z 296.32,A -85,B 0,C 180,E1 -21913.1,E2 -21913.1} C_VEL
LIN {X 0,Y 192.472,Z 296.321,A -85,B 0,C 180,E1 -21916.911,E2 -21916.911} C_VEL
LIN {X 0,Y 192.535,Z 296.311,A -85,B 0,C 180,E1 -21921.655,E2 -21921.655} C_VEL
LIN {X 0,Y 192.582,Z 296.304,A -85,B 0,C 180,E1 -21926.82,E2 -21926.82} C_VEL
LIN {X 0,Y 192.61,Z 296.305,A -85,B 0,C 180,E1 -21931.692,E2 -21931.692} C_VEL
LIN {X 0,Y 192.671,Z 296.285,A -85,B 0,C 180,E1 -21936.352,E2 -21936.352} C_VEL
LIN {X 0,Y 193.085,Z 296.224,A -85,B 0,C 180,E1 -21942.608,E2 -21942.608} C_VEL
LIN {X 0,Y 194.754,Z 312.82,A -85,B 0,C 180,E1 -21943.7,E2 -21943.7} C_VEL
LIN {X 0,Y 193.592,Z 367.84,A -85,B 0,C 180,E1 -21947.493,E2 -21947.493} C_VEL
LIN {X 0,Y 193.277,Z 379.205,A -85,B 0,C 180,E1 -21948.604,E2 -21948.604} C_VEL
LIN {X 0,Y 192.777,Z 390.603,A -85,B 0,C 180,E1 -21950.09,E2 -21950.09} C_VEL
LIN {X 0,Y 192.315,Z 400.774,A -85,B 0,C 180,E1 -21951.841,E2 -21951.841} C_VEL
LIN {X 0,Y 191.913,Z 409.43,A -85,B 0,C 180,E1 -21953.7,E2 -21953.7} C_VEL
LIN {X 0,Y 191.48,Z 419.337,A -85,B 0,C 180,E1 -21956.324,E2 -21956.324} C_VEL
LIN {X 0,Y 191.194,Z 427.107,A -85,B 0,C 180,E1 -21958.954,E2 -21958.954} C_VEL
LIN {X 0,Y 190.995,Z 433.457,A -85,B 0,C 180,E1 -21961.588,E2 -21961.588} C_VEL
LIN {X 0,Y 191.224,Z 438.624,A -85,B 0,C 180,E1 -21964.222,E2 -21964.222} C_VEL
LIN {X 0,Y 191.875,Z 443.544,A -85,B 0,C 180,E1 -21967.372,E2 -21967.372} C_VEL
LIN {X 0,Y 193.119,Z 447.365,A -85,B 0,C 180,E1 -21970.705,E2 -21970.705} C_VEL
LIN {X 0,Y 194.157,Z 448.961,A -85,B 0,C 180,E1 -21972.55,E2 -21972.55} C_VEL
LIN {X 0,Y 195.859,Z 450.243,A -85,B 0,C 180,E1 -21974.554,E2 -21974.554} C_VEL
LIN {X 0,Y 197.553,Z 451.105,A -85,B 0,C 180,E1 -21976.541,E2 -21976.541} C_VEL
LIN {X 0,Y 199.836,Z 451.545,A -85,B 0,C 180,E1 -21978.459,E2 -21978.459} C_VEL
LIN {X 0,Y 203.61,Z 451.221,A -85,B 0,C 180,E1 -21981.256,E2 -21981.256} C_VEL
LIN {X 0,Y 207.942,Z 449.831,A -85,B 0,C 180,E1 -21983.933,E2 -21983.933} C_VEL
LIN {X 0,Y 212.91,Z 447.362,A -85,B 0,C 180,E1 -21986.469,E2 -21986.469} C_VEL
LIN {X 0,Y 218.363,Z 443.717,A -85,B 0,C 180,E1 -21988.872,E2 -21988.872} C_VEL
LIN {X 0,Y 225.324,Z 437.775,A -85,B 0,C 180,E1 -21991.502,E2 -21991.502} C_VEL
LIN {X 0,Y 230.606,Z 432.256,A -85,B 0,C 180,E1 -21993.274,E2 -21993.274} C_VEL
LIN {X 0,Y 237.402,Z 424.024,A -85,B 0,C 180,E1 -21995.264,E2 -21995.264} C_VEL
LIN {X 0,Y 243.301,Z 415.241,A -85,B 0,C 180,E1 -21996.831,E2 -21996.831} C_VEL
LIN {X 0,Y 248.854,Z 405.49,A -85,B 0,C 180,E1 -21998.159,E2 -21998.159} C_VEL
LIN {X 0,Y 253.905,Z 394.61,A -85,B 0,C 180,E1 -21999.289,E2 -21999.289} C_VEL
LIN {X 0,Y 258.029,Z 383.433,A -85,B 0,C 180,E1 -22000.15,E2 -22000.15} C_VEL
LIN {X 0,Y 259.696,Z 377.756,A -85,B 0,C 180,E1 -22000.509,E2 -22000.509} C_VEL
LIN {X 0,Y 259.3,Z 376.514,A -85,B 0,C 180,E1 -22002.025,E2 -22002.025} C_VEL
LIN {X 0,Y 258.943,Z 376.66,A -85,B 0,C 180,E1 -22002.883,E2 -22002.883} C_VEL
LIN {X 0,Y 258.175,Z 378.504,A -85,B 0,C 180,E1 -22003.977,E2 -22003.977} C_VEL
LIN {X 0,Y 257.103,Z 382.157,A -85,B 0,C 180,E1 -22005.603,E2 -22005.603} C_VEL
LIN {X 0,Y 256.99,Z 383.173,A -85,B 0,C 180,E1 -22006.484,E2 -22006.484} C_VEL
LIN {X 0,Y 257.136,Z 384.107,A -85,B 0,C 180,E1 -22007.563,E2 -22007.563} C_VEL
LIN {X 0,Y 256.548,Z 386.016,A -85,B 0,C 180,E1 -22007.772,E2 -22007.772} C_VEL
LIN {X 0,Y 251.901,Z 398.055,A -85,B 0,C 180,E1 -22008.499,E2 -22008.499} C_VEL
LIN {X 0,Y 245.996,Z 410.015,A -85,B 0,C 180,E1 -22009.461,E2 -22009.461} C_VEL
LIN {X 0,Y 240.327,Z 419.625,A -85,B 0,C 180,E1 -22010.502,E2 -22010.502} C_VEL
LIN {X 0,Y 233.498,Z 429.361,A -85,B 0,C 180,E1 -22011.909,E2 -22011.909} C_VEL
LIN {X 0,Y 227.406,Z 436.688,A -85,B 0,C 180,E1 -22013.34,E2 -22013.34} C_VEL
LIN {X 0,Y 220.99,Z 443.453,A -85,B 0,C 180,E1 -22015.079,E2 -22015.079} C_VEL
LIN {X 0,Y 214.257,Z 449.609,A -85,B 0,C 180,E1 -22017.232,E2 -22017.232} C_VEL
LIN {X 0,Y 208.051,Z 454.368,A -85,B 0,C 180,E1 -22019.555,E2 -22019.555} C_VEL
LIN {X 0,Y 204.275,Z 456.809,A -85,B 0,C 180,E1 -22021.205,E2 -22021.205} C_VEL
LIN {X 0,Y 200.745,Z 458.744,A -85,B 0,C 180,E1 -22022.927,E2 -22022.927} C_VEL
LIN {X 0,Y 197.56,Z 460.247,A -85,B 0,C 180,E1 -22024.729,E2 -22024.729} C_VEL
LIN {X 0,Y 194.679,Z 461.35,A -85,B 0,C 180,E1 -22026.602,E2 -22026.602} C_VEL
LIN {X 0,Y 192.022,Z 461.921,A -85,B 0,C 180,E1 -22028.53,E2 -22028.53} C_VEL
LIN {X 0,Y 188.138,Z 461.85,A -85,B 0,C 180,E1 -22032.611,E2 -22032.611} C_VEL
LIN {X 0,Y 186.727,Z 461.21,A -85,B 0,C 180,E1 -22034.724,E2 -22034.724} C_VEL
LIN {X 0,Y 184.897,Z 458.501,A -85,B 0,C 180,E1 -22039.044,E2 -22039.044} C_VEL
LIN {X 0,Y 184.542,Z 455.774,A -85,B 0,C 180,E1 -22041.996,E2 -22041.996} C_VEL
LIN {X 0,Y 183.54,Z 460.719,A -85,B 0,C 180,E1 -22045.607,E2 -22045.607} C_VEL
LIN {X 0,Y 183.435,Z 462.965,A -85,B 0,C 180,E1 -22047.804,E2 -22047.804} C_VEL
LIN {X 0,Y 183.488,Z 464.574,A -85,B 0,C 180,E1 -22050,E2 -22050} C_VEL
LIN {X 0,Y 183.331,Z 465.617,A -85,B 0,C 180,E1 -22052.197,E2 -22052.197} C_VEL
LIN {X 0,Y 183.251,Z 466.189,A -85,B 0,C 180,E1 -22054.399,E2 -22054.399} C_VEL
LIN {X 0,Y 183.33,Z 466.311,A -85,B 0,C 180,E1 -22056.604,E2 -22056.604} C_VEL
LIN {X 0,Y 183.672,Z 465.927,A -85,B 0,C 180,E1 -22058.804,E2 -22058.804} C_VEL
LIN {X 0,Y 184.246,Z 464.974,A -85,B 0,C 180,E1 -22060.995,E2 -22060.995} C_VEL
LIN {X 0,Y 185.099,Z 463.558,A -85,B 0,C 180,E1 -22063.168,E2 -22063.168} C_VEL
LIN {X 0,Y 186.876,Z 460.492,A -85,B 0,C 180,E1 -22066.383,E2 -22066.383} C_VEL
LIN {X 0,Y 189.315,Z 456.179,A -85,B 0,C 180,E1 -22069.518,E2 -22069.518} C_VEL
LIN {X 0,Y 192.393,Z 450.262,A -85,B 0,C 180,E1 -22072.554,E2 -22072.554} C_VEL
LIN {X 0,Y 195.421,Z 443.966,A -85,B 0,C 180,E1 -22074.997,E2 -22074.997} C_VEL
LIN {X 0,Y 197.43,Z 439.522,A -85,B 0,C 180,E1 -22076.421,E2 -22076.421} C_VEL
LIN {X 0,Y 200.257,Z 432.414,A -85,B 0,C 180,E1 -22078.28,E2 -22078.28} C_VEL
LIN {X 0,Y 203.065,Z 424.497,A -85,B 0,C 180,E1 -22079.92,E2 -22079.92} C_VEL
LIN {X 0,Y 205.386,Z 417.111,A -85,B 0,C 180,E1 -22081.139,E2 -22081.139} C_VEL
LIN {X 0,Y 207.738,Z 408.198,A -85,B 0,C 180,E1 -22082.297,E2 -22082.297} C_VEL
LIN {X 0,Y 209.741,Z 399.395,A -85,B 0,C 180,E1 -22083.139,E2 -22083.139} C_VEL
LIN {X 0,Y 211.307,Z 389.829,A -85,B 0,C 180,E1 -22083.82,E2 -22083.82} C_VEL
LIN {X 0,Y 212.44,Z 378.269,A -85,B 0,C 180,E1 -22084.365,E2 -22084.365} C_VEL
LIN {X 0,Y 213.039,Z 364.031,A -85,B 0,C 180,E1 -22084.865,E2 -22084.865} C_VEL
LIN {X 0,Y 210.784,Z 347.284,A -85,B 0,C 180,E1 -22086.172,E2 -22086.172} C_VEL
LIN {X 0,Y 206.175,Z 336.472,A -85,B 0,C 180,E1 -22087.879,E2 -22087.879} C_VEL
LIN {X 0,Y 199.906,Z 323.94,A -85,B 0,C 180,E1 -22090.303,E2 -22090.303} C_VEL
LIN {X 0,Y 196.353,Z 317.914,A -85,B 0,C 180,E1 -22091.743,E2 -22091.743} C_VEL
LIN {X 0,Y 193.682,Z 313.406,A -85,B 0,C 180,E1 -22092.902,E2 -22092.902} C_VEL
LIN {X 0,Y 190.62,Z 308.455,A -85,B 0,C 180,E1 -22094.294,E2 -22094.294} C_VEL
LIN {X 0,Y 187.705,Z 304.24,A -85,B 0,C 180,E1 -22095.673,E2 -22095.673} C_VEL
LIN {X 0,Y 187.062,Z 302.807,A -85,B 0,C 180,E1 -22096.093,E2 -22096.093} C_VEL
LIN {X 0,Y 185.492,Z 297.182,A -85,B 0,C 180,E1 -22101.038,E2 -22101.038} C_VEL
LIN {X 0,Y 185.537,Z 297.183,A -85,B 0,C 180,E1 -22106.443,E2 -22106.443} C_VEL
LIN {X 0,Y 185.559,Z 297.178,A -85,B 0,C 180,E1 -22110.588,E2 -22110.588} C_VEL
LIN {X 0,Y 185.588,Z 297.177,A -85,B 0,C 180,E1 -22115.376,E2 -22115.376} C_VEL
LIN {X 0,Y 185.679,Z 297.167,A -85,B 0,C 180,E1 -22121.13,E2 -22121.13} C_VEL
LIN {X 0,Y 185.689,Z 297.152,A -85,B 0,C 180,E1 -22124.63,E2 -22124.63} C_VEL
LIN {X 0,Y 185.892,Z 297.121,A -85,B 0,C 180,E1 -22129.411,E2 -22129.411} C_VEL
LIN {X 0,Y 185.947,Z 297.116,A -85,B 0,C 180,E1 -22133.483,E2 -22133.483} C_VEL
LIN {X 0,Y 186.202,Z 297.095,A -85,B 0,C 180,E1 -22137.83,E2 -22137.83} C_VEL
LIN {X 0,Y 186.401,Z 297.057,A -85,B 0,C 180,E1 -22139.993,E2 -22139.993} C_VEL
LIN {X 0,Y 185.908,Z 297.124,A -85,B 0,C 180,E1 -22144.329,E2 -22144.329} C_VEL
LIN {X 0,Y 185.975,Z 297.128,A -85,B 0,C 180,E1 -22148.687,E2 -22148.687} C_VEL
LIN {X 0,Y 185.724,Z 297.164,A -85,B 0,C 180,E1 -22153.116,E2 -22153.116} C_VEL
LIN {X 0,Y 185.683,Z 297.166,A -85,B 0,C 180,E1 -22157.618,E2 -22157.618} C_VEL
LIN {X 0,Y 185.589,Z 297.179,A -85,B 0,C 180,E1 -22162.244,E2 -22162.244} C_VEL
LIN {X 0,Y 185.527,Z 297.189,A -85,B 0,C 180,E1 -22166.648,E2 -22166.648} C_VEL
LIN {X 0,Y 186.417,Z 299.825,A -85,B 0,C 180,E1 -22167.192,E2 -22167.192} C_VEL
LIN {X 0,Y 188.586,Z 302.123,A -85,B 0,C 180,E1 -22168.209,E2 -22168.209} C_VEL
LIN {X 0,Y 189.386,Z 302.946,A -85,B 0,C 180,E1 -22168.57,E2 -22168.57} C_VEL
LIN {X 0,Y 191.457,Z 306.202,A -85,B 0,C 180,E1 -22169.546,E2 -22169.546} C_VEL
LIN {X 0,Y 192.967,Z 307.909,A -85,B 0,C 180,E1 -22170.194,E2 -22170.194} C_VEL
LIN {X 0,Y 195.592,Z 311.556,A -85,B 0,C 180,E1 -22171.316,E2 -22171.316} C_VEL
LIN {X 0,Y 203.864,Z 323.903,A -85,B 0,C 180,E1 -22174.534,E2 -22174.534} C_VEL
LIN {X 0,Y 210.613,Z 335.454,A -85,B 0,C 180,E1 -22176.907,E2 -22176.907} C_VEL
LIN {X 0,Y 214.3,Z 342.886,A -85,B 0,C 180,E1 -22178.155,E2 -22178.155} C_VEL
LIN {X 0,Y 212.798,Z 368.664,A -85,B 0,C 180,E1 -22179.046,E2 -22179.046} C_VEL
LIN {X 0,Y 211.597,Z 379.695,A -85,B 0,C 180,E1 -22179.71,E2 -22179.71} C_VEL
LIN {X 0,Y 209.705,Z 390.398,A -85,B 0,C 180,E1 -22180.69,E2 -22180.69} C_VEL
LIN {X 0,Y 207.625,Z 399.638,A -85,B 0,C 180,E1 -22181.868,E2 -22181.868} C_VEL
LIN {X 0,Y 205.273,Z 407.915,A -85,B 0,C 180,E1 -22183.205,E2 -22183.205} C_VEL
LIN {X 0,Y 202.83,Z 415.423,A -85,B 0,C 180,E1 -22184.74,E2 -22184.74} C_VEL
LIN {X 0,Y 200.625,Z 421.374,A -85,B 0,C 180,E1 -22186.223,E2 -22186.223} C_VEL
LIN {X 0,Y 198.455,Z 426.46,A -85,B 0,C 180,E1 -22187.712,E2 -22187.712} C_VEL
LIN {X 0,Y 195.826,Z 432.12,A -85,B 0,C 180,E1 -22189.76,E2 -22189.76} C_VEL
LIN {X 0,Y 193.441,Z 436.79,A -85,B 0,C 180,E1 -22191.857,E2 -22191.857} C_VEL
LIN {X 0,Y 191.318,Z 440.626,A -85,B 0,C 180,E1 -22194.003,E2 -22194.003} C_VEL
LIN {X 0,Y 189.47,Z 443.721,A -85,B 0,C 180,E1 -22196.194,E2 -22196.194} C_VEL
LIN {X 0,Y 187.864,Z 446.104,A -85,B 0,C 180,E1 -22198.417,E2 -22198.417} C_VEL
LIN {X 0,Y 186.481,Z 447.835,A -85,B 0,C 180,E1 -22200.664,E2 -22200.664} C_VEL
LIN {X 0,Y 185.342,Z 449.002,A -85,B 0,C 180,E1 -22202.934,E2 -22202.934} C_VEL
LIN {X 0,Y 184.103,Z 449.779,A -85,B 0,C 180,E1 -22206.352,E2 -22206.352} C_VEL
LIN {X 0,Y 183.319,Z 449.338,A -85,B 0,C 180,E1 -22209.816,E2 -22209.816} C_VEL
LIN {X 0,Y 183.087,Z 448.311,A -85,B 0,C 180,E1 -22212.117,E2 -22212.117} C_VEL
LIN {X 0,Y 183.137,Z 445.786,A -85,B 0,C 180,E1 -22215.556,E2 -22215.556} C_VEL
LIN {X 0,Y 183.564,Z 441.848,A -85,B 0,C 180,E1 -22218.964,E2 -22218.964} C_VEL
LIN {X 0,Y 184.351,Z 436.513,A -85,B 0,C 180,E1 -22222.323,E2 -22222.323} C_VEL
LIN {X 0,Y 185.213,Z 430.762,A -85,B 0,C 180,E1 -22225.103,E2 -22225.103} C_VEL
LIN {X 0,Y 186.36,Z 423.449,A -85,B 0,C 180,E1 -22227.839,E2 -22227.839} C_VEL
LIN {X 0,Y 187.524,Z 416.158,A -85,B 0,C 180,E1 -22230,E2 -22230} C_VEL
LIN {X 0,Y 188.737,Z 408.373,A -85,B 0,C 180,E1 -22231.868,E2 -22231.868} C_VEL
LIN {X 0,Y 189.873,Z 400.538,A -85,B 0,C 180,E1 -22233.386,E2 -22233.386} C_VEL
LIN {X 0,Y 190.753,Z 393.567,A -85,B 0,C 180,E1 -22234.491,E2 -22234.491} C_VEL
LIN {X 0,Y 191.679,Z 384.212,A -85,B 0,C 180,E1 -22235.655,E2 -22235.655} C_VEL
LIN {X 0,Y 192.386,Z 374.968,A -85,B 0,C 180,E1 -22236.501,E2 -22236.501} C_VEL
LIN {X 0,Y 192.853,Z 365.047,A -85,B 0,C 180,E1 -22237.111,E2 -22237.111} C_VEL
LIN {X 0,Y 194.23,Z 319.272,A -85,B 0,C 180,E1 -22238.809,E2 -22238.809} C_VEL
LIN {X 0,Y 188.991,Z 304.869,A -85,B 0,C 180,E1 -22239.968,E2 -22239.968} C_VEL
LIN {X 0,Y 185.896,Z 297.483,A -85,B 0,C 180,E1 -22240.642,E2 -22240.642} C_VEL
LIN {X 0,Y 185.849,Z 297.149,A -85,B 0,C 180,E1 -22240.735,E2 -22240.735} C_VEL
LIN {X 0,Y 185.658,Z 297.171,A -85,B 0,C 180,E1 -22245.366,E2 -22245.366} C_VEL
LIN {X 0,Y 185.571,Z 297.181,A -85,B 0,C 180,E1 -22249.929,E2 -22249.929} C_VEL
LIN {X 0,Y 185.552,Z 297.185,A -85,B 0,C 180,E1 -22254.65,E2 -22254.65} C_VEL
LIN {X 0,Y 185.52,Z 297.184,A -85,B 0,C 180,E1 -22259.504,E2 -22259.504} C_VEL
LIN {X 0,Y 185.474,Z 297.19,A -85,B 0,C 180,E1 -22264.638,E2 -22264.638} C_VEL
LIN {X 0,Y 185.478,Z 297.192,A -85,B 0,C 180,E1 -22267.32,E2 -22267.32} C_VEL
LIN {X 0,Y 185.442,Z 297.195,A -85,B 0,C 180,E1 -22270.727,E2 -22270.727} C_VEL
LIN {X 0,Y 185.44,Z 297.198,A -85,B 0,C 180,E1 -22276.062,E2 -22276.062} C_VEL
LIN {X 0,Y 185.451,Z 297.193,A -85,B 0,C 180,E1 -22279.902,E2 -22279.902} C_VEL
LIN {X 0,Y 185.491,Z 297.19,A -85,B 0,C 180,E1 -22282.718,E2 -22282.718} C_VEL
LIN {X 0,Y 185.518,Z 297.185,A -85,B 0,C 180,E1 -22287.98,E2 -22287.98} C_VEL
LIN {X 0,Y 185.536,Z 297.185,A -85,B 0,C 180,E1 -22290.603,E2 -22290.603} C_VEL
LIN {X 0,Y 185.572,Z 297.175,A -85,B 0,C 180,E1 -22295.389,E2 -22295.389} C_VEL
LIN {X 0,Y 186.091,Z 297.096,A -85,B 0,C 180,E1 -22302.847,E2 -22302.847} C_VEL
LIN {X 0,Y 187.701,Z 312.986,A -85,B 0,C 180,E1 -22303.908,E2 -22303.908} C_VEL
LIN {X 0,Y 186.586,Z 367.869,A -85,B 0,C 180,E1 -22307.858,E2 -22307.858} C_VEL
LIN {X 0,Y 186.24,Z 380.115,A -85,B 0,C 180,E1 -22309.132,E2 -22309.132} C_VEL
LIN {X 0,Y 185.733,Z 391.677,A -85,B 0,C 180,E1 -22310.758,E2 -22310.758} C_VEL
LIN {X 0,Y 185.305,Z 401.921,A -85,B 0,C 180,E1 -22312.653,E2 -22312.653} C_VEL
LIN {X 0,Y 184.859,Z 411.421,A -85,B 0,C 180,E1 -22314.827,E2 -22314.827} C_VEL
LIN {X 0,Y 184.553,Z 420.082,A -85,B 0,C 180,E1 -22317.279,E2 -22317.279} C_VEL
LIN {X 0,Y 184.27,Z 426.37,A -85,B 0,C 180,E1 -22319.461,E2 -22319.461} C_VEL
LIN {X 0,Y 184.088,Z 432.77,A -85,B 0,C 180,E1 -22322.195,E2 -22322.195} C_VEL
LIN {X 0,Y 184.278,Z 437.13,A -85,B 0,C 180,E1 -22324.381,E2 -22324.381} C_VEL
LIN {X 0,Y 184.931,Z 442.416,A -85,B 0,C 180,E1 -22327.65,E2 -22327.65} C_VEL
LIN {X 0,Y 186.149,Z 446.533,A -85,B 0,C 180,E1 -22330.999,E2 -22330.999} C_VEL
LIN {X 0,Y 187.275,Z 448.449,A -85,B 0,C 180,E1 -22333.019,E2 -22333.019} C_VEL
LIN {X 0,Y 189.008,Z 450.08,A -85,B 0,C 180,E1 -22335.094,E2 -22335.094} C_VEL
LIN {X 0,Y 190.785,Z 451.225,A -85,B 0,C 180,E1 -22337.146,E2 -22337.146} C_VEL
LIN {X 0,Y 193.136,Z 451.825,A -85,B 0,C 180,E1 -22339.123,E2 -22339.123} C_VEL
LIN {X 0,Y 197.44,Z 451.946,A -85,B 0,C 180,E1 -22342.257,E2 -22342.257} C_VEL
LIN {X 0,Y 201.581,Z 451.067,A -85,B 0,C 180,E1 -22344.738,E2 -22344.738} C_VEL
LIN {X 0,Y 204.934,Z 449.798,A -85,B 0,C 180,E1 -22346.482,E2 -22346.482} C_VEL
LIN {X 0,Y 210.471,Z 447.065,A -85,B 0,C 180,E1 -22348.965,E2 -22348.965} C_VEL
LIN {X 0,Y 216.424,Z 443.133,A -85,B 0,C 180,E1 -22351.309,E2 -22351.309} C_VEL
LIN {X 0,Y 222.837,Z 437.761,A -85,B 0,C 180,E1 -22353.505,E2 -22353.505} C_VEL
LIN {X 0,Y 228.527,Z 432.188,A -85,B 0,C 180,E1 -22355.219,E2 -22355.219} C_VEL
LIN {X 0,Y 234.493,Z 425.304,A -85,B 0,C 180,E1 -22356.834,E2 -22356.834} C_VEL
LIN {X 0,Y 240.704,Z 416.894,A -85,B 0,C 180,E1 -22358.354,E2 -22358.354} C_VEL
LIN {X 0,Y 246.238,Z 407.837,A -85,B 0,C 180,E1 -22359.59,E2 -22359.59} C_VEL
LIN {X 0,Y 252.056,Z 396.361,A -85,B 0,C 180,E1 -22360.79,E2 -22360.79} C_VEL
LIN {X 0,Y 256.353,Z 385.606,A -85,B 0,C 180,E1 -22361.611,E2 -22361.611} C_VEL
LIN {X 0,Y 256.863,Z 384.195,A -85,B 0,C 180,E1 -22361.703,E2 -22361.703} C_VEL
LIN {X 0,Y 257.088,Z 383.451,A -85,B 0,C 180,E1 -22361.851,E2 -22361.851} C_VEL
LIN {X 0,Y 256.951,Z 382.676,A -85,B 0,C 180,E1 -22363.145,E2 -22363.145} C_VEL
LIN {X 0,Y 256.88,Z 382.634,A -85,B 0,C 180,E1 -22365.349,E2 -22365.349} C_VEL
LIN {X 0,Y 256.99,Z 383.173,A -85,B 0,C 180,E1 -22366.484,E2 -22366.484} C_VEL
LIN {X 0,Y 256.798,Z 384.11,A -85,B 0,C 180,E1 -22366.866,E2 -22366.866} C_VEL
LIN {X 0,Y 256.06,Z 386.365,A -85,B 0,C 180,E1 -22367.151,E2 -22367.151} C_VEL
LIN {X 0,Y 254.648,Z 390.194,A -85,B 0,C 180,E1 -22367.268,E2 -22367.268} C_VEL
LIN {X 0,Y 250.106,Z 399.946,A -85,B 0,C 180,E1 -22367.067,E2 -22367.067} C_VEL
LIN {X 0,Y 248.733,Z 402.568,A -85,B 0,C 180,E1 -22367.176,E2 -22367.176} C_VEL
LIN {X 0,Y 243.113,Z 412.871,A -85,B 0,C 180,E1 -22368.048,E2 -22368.048} C_VEL
LIN {X 0,Y 236.53,Z 422.798,A -85,B 0,C 180,E1 -22369.18,E2 -22369.18} C_VEL
LIN {X 0,Y 229.649,Z 431.505,A -85,B 0,C 180,E1 -22370.515,E2 -22370.515} C_VEL
LIN {X 0,Y 223.556,Z 438.217,A -85,B 0,C 180,E1 -22371.875,E2 -22371.875} C_VEL
LIN {X 0,Y 215.354,Z 445.906,A -85,B 0,C 180,E1 -22374.025,E2 -22374.025} C_VEL
LIN {X 0,Y 208.412,Z 451.318,A -85,B 0,C 180,E1 -22376.192,E2 -22376.192} C_VEL
LIN {X 0,Y 202.014,Z 455.468,A -85,B 0,C 180,E1 -22378.543,E2 -22378.543} C_VEL
LIN {X 0,Y 198.109,Z 457.603,A -85,B 0,C 180,E1 -22380.22,E2 -22380.22} C_VEL
LIN {X 0,Y 194.468,Z 459.308,A -85,B 0,C 180,E1 -22381.977,E2 -22381.977} C_VEL
LIN {X 0,Y 191.182,Z 460.482,A -85,B 0,C 180,E1 -22383.824,E2 -22383.824} C_VEL
LIN {X 0,Y 185.45,Z 461.554,A -85,B 0,C 180,E1 -22387.73,E2 -22387.73} C_VEL
LIN {X 0,Y 183.199,Z 461.509,A -85,B 0,C 180,E1 -22389.802,E2 -22389.802} C_VEL
LIN {X 0,Y 179.981,Z 460.049,A -85,B 0,C 180,E1 -22394.136,E2 -22394.136} C_VEL
LIN {X 0,Y 178.842,Z 458.788,A -85,B 0,C 180,E1 -22396.362,E2 -22396.362} C_VEL
LIN {X 0,Y 177.875,Z 455.914,A -85,B 0,C 180,E1 -22399.758,E2 -22399.758} C_VEL
LIN {X 0,Y 177.747,Z 454.446,A -85,B 0,C 180,E1 -22401.33,E2 -22401.33} C_VEL
LIN {X 0,Y 176.672,Z 458.601,A -85,B 0,C 180,E1 -22404.178,E2 -22404.178} C_VEL
LIN {X 0,Y 176.362,Z 462.426,A -85,B 0,C 180,E1 -22407.716,E2 -22407.716} C_VEL
LIN {X 0,Y 176.425,Z 464.073,A -85,B 0,C 180,E1 -22410,E2 -22410} C_VEL
LIN {X 0,Y 176.153,Z 465.763,A -85,B 0,C 180,E1 -22414.037,E2 -22414.037} C_VEL
LIN {X 0,Y 176.265,Z 466.014,A -85,B 0,C 180,E1 -22416.869,E2 -22416.869} C_VEL
LIN {X 0,Y 176.642,Z 465.639,A -85,B 0,C 180,E1 -22419.157,E2 -22419.157} C_VEL
LIN {X 0,Y 177.268,Z 464.755,A -85,B 0,C 180,E1 -22421.433,E2 -22421.433} C_VEL
LIN {X 0,Y 178.17,Z 463.416,A -85,B 0,C 180,E1 -22423.69,E2 -22423.69} C_VEL
LIN {X 0,Y 180.055,Z 460.43,A -85,B 0,C 180,E1 -22427.022,E2 -22427.022} C_VEL
LIN {X 0,Y 181.691,Z 457.738,A -85,B 0,C 180,E1 -22429.195,E2 -22429.195} C_VEL
LIN {X 0,Y 184.731,Z 452.525,A -85,B 0,C 180,E1 -22432.361,E2 -22432.361} C_VEL
LIN {X 0,Y 188.378,Z 445.702,A -85,B 0,C 180,E1 -22435.406,E2 -22435.406} C_VEL
LIN {X 0,Y 191.747,Z 438.288,A -85,B 0,C 180,E1 -22437.86,E2 -22437.86} C_VEL
LIN {X 0,Y 194.891,Z 430.988,A -85,B 0,C 180,E1 -22439.725,E2 -22439.725} C_VEL
LIN {X 0,Y 197.463,Z 423.863,A -85,B 0,C 180,E1 -22441.21,E2 -22441.21} C_VEL
LIN {X 0,Y 200.144,Z 415.61,A -85,B 0,C 180,E1 -22442.559,E2 -22442.559} C_VEL
LIN {X 0,Y 202.63,Z 406.51,A -85,B 0,C 180,E1 -22443.706,E2 -22443.706} C_VEL
LIN {X 0,Y 205.096,Z 395.319,A -85,B 0,C 180,E1 -22444.723,E2 -22444.723} C_VEL
LIN {X 0,Y 206.621,Z 383.896,A -85,B 0,C 180,E1 -22445.401,E2 -22445.401} C_VEL
LIN {X 0,Y 207.71,Z 365.173,A -85,B 0,C 180,E1 -22446.107,E2 -22446.107} C_VEL
LIN {X 0,Y 205.742,Z 350.061,A -85,B 0,C 180,E1 -22447.335,E2 -22447.335} C_VEL
LIN {X 0,Y 201.335,Z 339.859,A -85,B 0,C 180,E1 -22449.059,E2 -22449.059} C_VEL
LIN {X 0,Y 196.051,Z 328.97,A -85,B 0,C 180,E1 -22451.232,E2 -22451.232} C_VEL
LIN {X 0,Y 192.096,Z 322.057,A -85,B 0,C 180,E1 -22452.962,E2 -22452.962} C_VEL
LIN {X 0,Y 189.617,Z 317.94,A -85,B 0,C 180,E1 -22454.103,E2 -22454.103} C_VEL
LIN {X 0,Y 187.221,Z 313.886,A -85,B 0,C 180,E1 -22455.265,E2 -22455.265} C_VEL
LIN {X 0,Y 184.183,Z 309.203,A -85,B 0,C 180,E1 -22456.8,E2 -22456.8} C_VEL
LIN {X 0,Y 180.345,Z 303.685,A -85,B 0,C 180,E1 -22458.874,E2 -22458.874} C_VEL
LIN {X 0,Y 179.669,Z 302.247,A -85,B 0,C 180,E1 -22459.335,E2 -22459.335} C_VEL
LIN {X 0,Y 178.441,Z 298.064,A -85,B 0,C 180,E1 -22463.522,E2 -22463.522} C_VEL
LIN {X 0,Y 178.493,Z 298.061,A -85,B 0,C 180,E1 -22466.541,E2 -22466.541} C_VEL
LIN {X 0,Y 178.458,Z 298.066,A -85,B 0,C 180,E1 -22471.791,E2 -22471.791} C_VEL
LIN {X 0,Y 178.524,Z 298.051,A -85,B 0,C 180,E1 -22474.883,E2 -22474.883} C_VEL
LIN {X 0,Y 178.627,Z 298.046,A -85,B 0,C 180,E1 -22480.781,E2 -22480.781} C_VEL
LIN {X 0,Y 178.656,Z 298.04,A -85,B 0,C 180,E1 -22486.341,E2 -22486.341} C_VEL
LIN {X 0,Y 178.915,Z 298,A -85,B 0,C 180,E1 -22490.953,E2 -22490.953} C_VEL
LIN {X 0,Y 179.148,Z 297.974,A -85,B 0,C 180,E1 -22497.745,E2 -22497.745} C_VEL
LIN {X 0,Y 179.365,Z 297.933,A -85,B 0,C 180,E1 -22499.993,E2 -22499.993} C_VEL
LIN {X 0,Y 178.855,Z 298.001,A -85,B 0,C 180,E1 -22504.5,E2 -22504.5} C_VEL
LIN {X 0,Y 178.904,Z 298.005,A -85,B 0,C 180,E1 -22509.033,E2 -22509.033} C_VEL
LIN {X 0,Y 178.652,Z 298.043,A -85,B 0,C 180,E1 -22513.645,E2 -22513.645} C_VEL
LIN {X 0,Y 178.615,Z 298.041,A -85,B 0,C 180,E1 -22519.209,E2 -22519.209} C_VEL
LIN {X 0,Y 178.506,Z 298.056,A -85,B 0,C 180,E1 -22523.496,E2 -22523.496} C_VEL
LIN {X 0,Y 179.37,Z 300.661,A -85,B 0,C 180,E1 -22524.119,E2 -22524.119} C_VEL
LIN {X 0,Y 181.62,Z 303.081,A -85,B 0,C 180,E1 -22525.337,E2 -22525.337} C_VEL
LIN {X 0,Y 182.448,Z 303.677,A -85,B 0,C 180,E1 -22525.748,E2 -22525.748} C_VEL
LIN {X 0,Y 184.192,Z 306.675,A -85,B 0,C 180,E1 -22526.704,E2 -22526.704} C_VEL
LIN {X 0,Y 186.295,Z 308.934,A -85,B 0,C 180,E1 -22527.721,E2 -22527.721} C_VEL
LIN {X 0,Y 188.808,Z 312.493,A -85,B 0,C 180,E1 -22528.931,E2 -22528.931} C_VEL
LIN {X 0,Y 190.166,Z 314.387,A -85,B 0,C 180,E1 -22529.558,E2 -22529.558} C_VEL
LIN {X 0,Y 193.446,Z 319.074,A -85,B 0,C 180,E1 -22531.008,E2 -22531.008} C_VEL
LIN {X 0,Y 200.135,Z 329.247,A -85,B 0,C 180,E1 -22533.721,E2 -22533.721} C_VEL
LIN {X 0,Y 206.797,Z 341.026,A -85,B 0,C 180,E1 -22536.183,E2 -22536.183} C_VEL
LIN {X 0,Y 208.827,Z 344.944,A -85,B 0,C 180,E1 -22536.898,E2 -22536.898} C_VEL
LIN {X 0,Y 207.443,Z 369.116,A -85,B 0,C 180,E1 -22537.778,E2 -22537.778} C_VEL
LIN {X 0,Y 206.276,Z 379.446,A -85,B 0,C 180,E1 -22538.406,E2 -22538.406} C_VEL
LIN {X 0,Y 204.45,Z 389.815,A -85,B 0,C 180,E1 -22539.337,E2 -22539.337} C_VEL
LIN {X 0,Y 202.256,Z 399.241,A -85,B 0,C 180,E1 -22540.527,E2 -22540.527} C_VEL
LIN {X 0,Y 199.597,Z 408.189,A -85,B 0,C 180,E1 -22541.98,E2 -22541.98} C_VEL
LIN {X 0,Y 197.242,Z 415.263,A -85,B 0,C 180,E1 -22543.449,E2 -22543.449} C_VEL
LIN {X 0,Y 194.521,Z 422.185,A -85,B 0,C 180,E1 -22545.209,E2 -22545.209} C_VEL
LIN {X 0,Y 191.73,Z 428.331,A -85,B 0,C 180,E1 -22547.136,E2 -22547.136} C_VEL
LIN {X 0,Y 188.844,Z 434.005,A -85,B 0,C 180,E1 -22549.363,E2 -22549.363} C_VEL
LIN {X 0,Y 186.397,Z 438.385,A -85,B 0,C 180,E1 -22551.529,E2 -22551.529} C_VEL
LIN {X 0,Y 184.142,Z 442.11,A -85,B 0,C 180,E1 -22553.863,E2 -22553.863} C_VEL
LIN {X 0,Y 181.509,Z 446.004,A -85,B 0,C 180,E1 -22557.175,E2 -22557.175} C_VEL
LIN {X 0,Y 179.981,Z 447.864,A -85,B 0,C 180,E1 -22559.494,E2 -22559.494} C_VEL
LIN {X 0,Y 178.692,Z 449.158,A -85,B 0,C 180,E1 -22561.839,E2 -22561.839} C_VEL
LIN {X 0,Y 177.143,Z 450.113,A -85,B 0,C 180,E1 -22565.831,E2 -22565.831} C_VEL
LIN {X 0,Y 176.346,Z 449.777,A -85,B 0,C 180,E1 -22568.981,E2 -22568.981} C_VEL
LIN {X 0,Y 176.049,Z 448.835,A -85,B 0,C 180,E1 -22571.376,E2 -22571.376} C_VEL
LIN {X 0,Y 176.004,Z 446.505,A -85,B 0,C 180,E1 -22574.957,E2 -22574.957} C_VEL
LIN {X 0,Y 176.388,Z 442.764,A -85,B 0,C 180,E1 -22578.509,E2 -22578.509} C_VEL
LIN {X 0,Y 176.831,Z 439.535,A -85,B 0,C 180,E1 -22580.853,E2 -22580.853} C_VEL
LIN {X 0,Y 177.665,Z 434.385,A -85,B 0,C 180,E1 -22583.755,E2 -22583.755} C_VEL
LIN {X 0,Y 178.414,Z 429.387,A -85,B 0,C 180,E1 -22586.048,E2 -22586.048} C_VEL
LIN {X 0,Y 179.432,Z 423.33,A -85,B 0,C 180,E1 -22588.317,E2 -22588.317} C_VEL
LIN {X 0,Y 180.661,Z 415.949,A -85,B 0,C 180,E1 -22590.558,E2 -22590.558} C_VEL
LIN {X 0,Y 181.727,Z 409.311,A -85,B 0,C 180,E1 -22592.217,E2 -22592.217} C_VEL
LIN {X 0,Y 183.008,Z 400.936,A -85,B 0,C 180,E1 -22593.91,E2 -22593.91} C_VEL
LIN {X 0,Y 184.04,Z 392.921,A -85,B 0,C 180,E1 -22595.204,E2 -22595.204} C_VEL
LIN {X 0,Y 184.884,Z 384.512,A -85,B 0,C 180,E1 -22596.275,E2 -22596.275} C_VEL
LIN {X 0,Y 185.634,Z 375.358,A -85,B 0,C 180,E1 -22597.139,E2 -22597.139} C_VEL
LIN {X 0,Y 186.113,Z 365.367,A -85,B 0,C 180,E1 -22597.777,E2 -22597.777} C_VEL
LIN {X 0,Y 187.564,Z 320.774,A -85,B 0,C 180,E1 -22599.484,E2 -22599.484} C_VEL
LIN {X 0,Y 182.732,Z 307.56,A -85,B 0,C 180,E1 -22600.608,E2 -22600.608} C_VEL
LIN {X 0,Y 178.882,Z 298.837,A -85,B 0,C 180,E1 -22601.471,E2 -22601.471} C_VEL
LIN {X 0,Y 178.718,Z 298.031,A -85,B 0,C 180,E1 -22601.573,E2 -22601.573} C_VEL
LIN {X 0,Y 178.585,Z 298.05,A -85,B 0,C 180,E1 -22605.991,E2 -22605.991} C_VEL
LIN {X 0,Y 178.594,Z 298.052,A -85,B 0,C 180,E1 -22609.217,E2 -22609.217} C_VEL
LIN {X 0,Y 178.49,Z 298.066,A -85,B 0,C 180,E1 -22615.115,E2 -22615.115} C_VEL
LIN {X 0,Y 178.436,Z 298.062,A -85,B 0,C 180,E1 -22620.799,E2 -22620.799} C_VEL
LIN {X 0,Y 178.46,Z 298.064,A -85,B 0,C 180,E1 -22624.223,E2 -22624.223} C_VEL
LIN {X 0,Y 178.367,Z 298.073,A -85,B 0,C 180,E1 -22629.083,E2 -22629.083} C_VEL
LIN {X 0,Y 178.374,Z 298.076,A -85,B 0,C 180,E1 -22632.053,E2 -22632.053} C_VEL
LIN {X 0,Y 178.374,Z 298.074,A -85,B 0,C 180,E1 -22635.171,E2 -22635.171} C_VEL
LIN {X 0,Y 178.386,Z 298.075,A -85,B 0,C 180,E1 -22638.466,E2 -22638.466} C_VEL
LIN {X 0,Y 178.408,Z 298.075,A -85,B 0,C 180,E1 -22643.79,E2 -22643.79} C_VEL
LIN {X 0,Y 178.471,Z 298.062,A -85,B 0,C 180,E1 -22646.553,E2 -22646.553} C_VEL
LIN {X 0,Y 178.433,Z 298.072,A -85,B 0,C 180,E1 -22651.803,E2 -22651.803} C_VEL
LIN {X 0,Y 178.503,Z 298.047,A -85,B 0,C 180,E1 -22656.823,E2 -22656.823} C_VEL
LIN {X 0,Y 179.093,Z 297.969,A -85,B 0,C 180,E1 -22663.039,E2 -22663.039} C_VEL
LIN {X 0,Y 180.645,Z 313.051,A -85,B 0,C 180,E1 -22664.132,E2 -22664.132} C_VEL
LIN {X 0,Y 179.601,Z 367.999,A -85,B 0,C 180,E1 -22668.341,E2 -22668.341} C_VEL
LIN {X 0,Y 179.301,Z 379.845,A -85,B 0,C 180,E1 -22669.614,E2 -22669.614} C_VEL
LIN {X 0,Y 178.812,Z 391.205,A -85,B 0,C 180,E1 -22671.247,E2 -22671.247} C_VEL
LIN {X 0,Y 178.379,Z 401.611,A -85,B 0,C 180,E1 -22673.219,E2 -22673.219} C_VEL
LIN {X 0,Y 177.985,Z 410.073,A -85,B 0,C 180,E1 -22675.194,E2 -22675.194} C_VEL
LIN {X 0,Y 177.693,Z 418.957,A -85,B 0,C 180,E1 -22677.741,E2 -22677.741} C_VEL
LIN {X 0,Y 177.331,Z 426.783,A -85,B 0,C 180,E1 -22680.575,E2 -22680.575} C_VEL
LIN {X 0,Y 177.262,Z 433.183,A -85,B 0,C 180,E1 -22683.417,E2 -22683.417} C_VEL
LIN {X 0,Y 177.546,Z 437.509,A -85,B 0,C 180,E1 -22685.686,E2 -22685.686} C_VEL
LIN {X 0,Y 178.345,Z 442.702,A -85,B 0,C 180,E1 -22689.076,E2 -22689.076} C_VEL
LIN {X 0,Y 179.75,Z 446.748,A -85,B 0,C 180,E1 -22692.424,E2 -22692.424} C_VEL
LIN {X 0,Y 182.172,Z 449.7,A -85,B 0,C 180,E1 -22695.674,E2 -22695.674} C_VEL
LIN {X 0,Y 184.015,Z 451.039,A -85,B 0,C 180,E1 -22697.797,E2 -22697.797} C_VEL
LIN {X 0,Y 186.452,Z 451.993,A -85,B 0,C 180,E1 -22699.837,E2 -22699.837} C_VEL
LIN {X 0,Y 189.06,Z 452.513,A -85,B 0,C 180,E1 -22701.829,E2 -22701.829} C_VEL
LIN {X 0,Y 191.983,Z 452.478,A -85,B 0,C 180,E1 -22703.752,E2 -22703.752} C_VEL
LIN {X 0,Y 195.202,Z 452.009,A -85,B 0,C 180,E1 -22705.604,E2 -22705.604} C_VEL
LIN {X 0,Y 198.706,Z 451.129,A -85,B 0,C 180,E1 -22707.38,E2 -22707.38} C_VEL
LIN {X 0,Y 202.455,Z 449.789,A -85,B 0,C 180,E1 -22709.084,E2 -22709.084} C_VEL
LIN {X 0,Y 208.493,Z 446.723,A -85,B 0,C 180,E1 -22711.505,E2 -22711.505} C_VEL
LIN {X 0,Y 215.032,Z 442.45,A -85,B 0,C 180,E1 -22713.759,E2 -22713.759} C_VEL
LIN {X 0,Y 221.936,Z 436.845,A -85,B 0,C 180,E1 -22715.868,E2 -22715.868} C_VEL
LIN {X 0,Y 229.318,Z 429.677,A -85,B 0,C 180,E1 -22717.808,E2 -22717.808} C_VEL
LIN {X 0,Y 236.058,Z 421.589,A -85,B 0,C 180,E1 -22719.408,E2 -22719.408} C_VEL
LIN {X 0,Y 242.564,Z 412.504,A -85,B 0,C 180,E1 -22720.769,E2 -22720.769} C_VEL
LIN {X 0,Y 248.372,Z 402.405,A -85,B 0,C 180,E1 -22721.913,E2 -22721.913} C_VEL
LIN {X 0,Y 252.901,Z 392.881,A -85,B 0,C 180,E1 -22722.734,E2 -22722.734} C_VEL
LIN {X 0,Y 254.288,Z 389.647,A -85,B 0,C 180,E1 -22722.977,E2 -22722.977} C_VEL
LIN {X 0,Y 254.319,Z 389.259,A -85,B 0,C 180,E1 -22724.069,E2 -22724.069} C_VEL
LIN {X 0,Y 254.453,Z 389.744,A -85,B 0,C 180,E1 -22726.33,E2 -22726.33} C_VEL
LIN {X 0,Y 248.733,Z 402.568,A -85,B 0,C 180,E1 -22727.176,E2 -22727.176} C_VEL
LIN {X 0,Y 246.814,Z 406.192,A -85,B 0,C 180,E1 -22727.288,E2 -22727.288} C_VEL
LIN {X 0,Y 239.327,Z 417.258,A -85,B 0,C 180,E1 -22726.918,E2 -22726.918} C_VEL
LIN {X 0,Y 237.059,Z 420.38,A -85,B 0,C 180,E1 -22727.107,E2 -22727.107} C_VEL
LIN {X 0,Y 229.898,Z 429.361,A -85,B 0,C 180,E1 -22728.325,E2 -22728.325} C_VEL
LIN {X 0,Y 222.811,Z 436.88,A -85,B 0,C 180,E1 -22729.712,E2 -22729.712} C_VEL
LIN {X 0,Y 214.843,Z 444.197,A -85,B 0,C 180,E1 -22731.571,E2 -22731.571} C_VEL
LIN {X 0,Y 207.34,Z 449.843,A -85,B 0,C 180,E1 -22733.616,E2 -22733.616} C_VEL
LIN {X 0,Y 200.344,Z 454.202,A -85,B 0,C 180,E1 -22735.855,E2 -22735.855} C_VEL
LIN {X 0,Y 196.044,Z 456.514,A -85,B 0,C 180,E1 -22737.47,E2 -22737.47} C_VEL
LIN {X 0,Y 191.997,Z 458.292,A -85,B 0,C 180,E1 -22739.171,E2 -22739.171} C_VEL
LIN {X 0,Y 188.246,Z 459.581,A -85,B 0,C 180,E1 -22740.964,E2 -22740.964} C_VEL
LIN {X 0,Y 181.773,Z 461.022,A -85,B 0,C 180,E1 -22744.83,E2 -22744.83} C_VEL
LIN {X 0,Y 178.92,Z 461.01,A -85,B 0,C 180,E1 -22746.871,E2 -22746.871} C_VEL
LIN {X 0,Y 174.747,Z 459.978,A -85,B 0,C 180,E1 -22751.231,E2 -22751.231} C_VEL
LIN {X 0,Y 173.265,Z 458.791,A -85,B 0,C 180,E1 -22753.504,E2 -22753.504} C_VEL
LIN {X 0,Y 171.371,Z 455.225,A -85,B 0,C 180,E1 -22758.167,E2 -22758.167} C_VEL
LIN {X 0,Y 171.015,Z 452.983,A -85,B 0,C 180,E1 -22760.538,E2 -22760.538} C_VEL
LIN {X 0,Y 169.609,Z 458.045,A -85,B 0,C 180,E1 -22764.026,E2 -22764.026} C_VEL
LIN {X 0,Y 169.292,Z 461.846,A -85,B 0,C 180,E1 -22767.62,E2 -22767.62} C_VEL
LIN {X 0,Y 169.362,Z 463.561,A -85,B 0,C 180,E1 -22770,E2 -22770} C_VEL
LIN {X 0,Y 169.071,Z 465.293,A -85,B 0,C 180,E1 -22773.854,E2 -22773.854} C_VEL
LIN {X 0,Y 169.225,Z 465.695,A -85,B 0,C 180,E1 -22777.157,E2 -22777.157} C_VEL
LIN {X 0,Y 169.634,Z 465.348,A -85,B 0,C 180,E1 -22779.539,E2 -22779.539} C_VEL
LIN {X 0,Y 170.31,Z 464.538,A -85,B 0,C 180,E1 -22781.907,E2 -22781.907} C_VEL
LIN {X 0,Y 171.265,Z 463.274,A -85,B 0,C 180,E1 -22784.253,E2 -22784.253} C_VEL
LIN {X 0,Y 173.265,Z 460.368,A -85,B 0,C 180,E1 -22787.711,E2 -22787.711} C_VEL
LIN {X 0,Y 175.98,Z 456.229,A -85,B 0,C 180,E1 -22791.065,E2 -22791.065} C_VEL
LIN {X 0,Y 179.401,Z 450.672,A -85,B 0,C 180,E1 -22794.288,E2 -22794.288} C_VEL
LIN {X 0,Y 182.673,Z 444.62,A -85,B 0,C 180,E1 -22796.875,E2 -22796.875} C_VEL
LIN {X 0,Y 185.515,Z 438.746,A -85,B 0,C 180,E1 -22798.882,E2 -22798.882} C_VEL
LIN {X 0,Y 188.788,Z 431.602,A -85,B 0,C 180,E1 -22800.788,E2 -22800.788} C_VEL
LIN {X 0,Y 191.468,Z 424.667,A -85,B 0,C 180,E1 -22802.303,E2 -22802.303} C_VEL
LIN {X 0,Y 194.269,Z 416.532,A -85,B 0,C 180,E1 -22803.7,E2 -22803.7} C_VEL
LIN {X 0,Y 196.766,Z 407.911,A -85,B 0,C 180,E1 -22804.853,E2 -22804.853} C_VEL
LIN {X 0,Y 199.011,Z 398.732,A -85,B 0,C 180,E1 -22805.756,E2 -22805.756} C_VEL
LIN {X 0,Y 200.789,Z 388.307,A -85,B 0,C 180,E1 -22806.514,E2 -22806.514} C_VEL
LIN {X 0,Y 202.109,Z 374.4,A -85,B 0,C 180,E1 -22807.118,E2 -22807.118} C_VEL
LIN {X 0,Y 202.457,Z 366.302,A -85,B 0,C 180,E1 -22807.422,E2 -22807.422} C_VEL
LIN {X 0,Y 200.777,Z 352.981,A -85,B 0,C 180,E1 -22808.552,E2 -22808.552} C_VEL
LIN {X 0,Y 195.405,Z 340.599,A -85,B 0,C 180,E1 -22810.805,E2 -22810.805} C_VEL
LIN {X 0,Y 191.131,Z 331.936,A -85,B 0,C 180,E1 -22812.727,E2 -22812.727} C_VEL
LIN {X 0,Y 186.378,Z 323.52,A -85,B 0,C 180,E1 -22814.996,E2 -22814.996} C_VEL
LIN {X 0,Y 183.722,Z 319.088,A -85,B 0,C 180,E1 -22816.351,E2 -22816.351} C_VEL
LIN {X 0,Y 180.098,Z 313.408,A -85,B 0,C 180,E1 -22818.311,E2 -22818.311} C_VEL
LIN {X 0,Y 177.125,Z 308.792,A -85,B 0,C 180,E1 -22820.055,E2 -22820.055} C_VEL
LIN {X 0,Y 172.769,Z 302.847,A -85,B 0,C 180,E1 -22822.848,E2 -22822.848} C_VEL
LIN {X 0,Y 172.187,Z 301.572,A -85,B 0,C 180,E1 -22823.343,E2 -22823.343} C_VEL
LIN {X 0,Y 171.458,Z 298.935,A -85,B 0,C 180,E1 -22826.395,E2 -22826.395} C_VEL
LIN {X 0,Y 171.421,Z 298.938,A -85,B 0,C 180,E1 -22830.522,E2 -22830.522} C_VEL
LIN {X 0,Y 171.449,Z 298.941,A -85,B 0,C 180,E1 -22835.793,E2 -22835.793} C_VEL
LIN {X 0,Y 171.583,Z 298.923,A -85,B 0,C 180,E1 -22840.865,E2 -22840.865} C_VEL
LIN {X 0,Y 171.573,Z 298.919,A -85,B 0,C 180,E1 -22845.765,E2 -22845.765} C_VEL
LIN {X 0,Y 171.852,Z 298.876,A -85,B 0,C 180,E1 -22850.578,E2 -22850.578} C_VEL
LIN {X 0,Y 171.808,Z 298.875,A -85,B 0,C 180,E1 -22855.3,E2 -22855.3} C_VEL
LIN {X 0,Y 172.328,Z 298.809,A -85,B 0,C 180,E1 -22859.992,E2 -22859.992} C_VEL
LIN {X 0,Y 171.803,Z 298.878,A -85,B 0,C 180,E1 -22864.685,E2 -22864.685} C_VEL
LIN {X 0,Y 171.842,Z 298.88,A -85,B 0,C 180,E1 -22869.407,E2 -22869.407} C_VEL
LIN {X 0,Y 171.569,Z 298.919,A -85,B 0,C 180,E1 -22874.22,E2 -22874.22} C_VEL
LIN {X 0,Y 171.535,Z 298.919,A -85,B 0,C 180,E1 -22879.739,E2 -22879.739} C_VEL
LIN {X 0,Y 172.355,Z 301.507,A -85,B 0,C 180,E1 -22880.474,E2 -22880.474} C_VEL
LIN {X 0,Y 174.261,Z 303.754,A -85,B 0,C 180,E1 -22881.74,E2 -22881.74} C_VEL
LIN {X 0,Y 175.756,Z 304.867,A -85,B 0,C 180,E1 -22882.627,E2 -22882.627} C_VEL
LIN {X 0,Y 177.674,Z 307.996,A -85,B 0,C 180,E1 -22883.827,E2 -22883.827} C_VEL
LIN {X 0,Y 179.777,Z 310.173,A -85,B 0,C 180,E1 -22884.984,E2 -22884.984} C_VEL
LIN {X 0,Y 182.327,Z 313.706,A -85,B 0,C 180,E1 -22886.372,E2 -22886.372} C_VEL
LIN {X 0,Y 183.756,Z 315.618,A -85,B 0,C 180,E1 -22887.109,E2 -22887.109} C_VEL
LIN {X 0,Y 187.39,Z 320.716,A -85,B 0,C 180,E1 -22888.894,E2 -22888.894} C_VEL
LIN {X 0,Y 191.842,Z 327.289,A -85,B 0,C 180,E1 -22890.923,E2 -22890.923} C_VEL
LIN {X 0,Y 197.775,Z 336.945,A -85,B 0,C 180,E1 -22893.412,E2 -22893.412} C_VEL
LIN {X 0,Y 203.561,Z 347.577,A -85,B 0,C 180,E1 -22895.63,E2 -22895.63} C_VEL
LIN {X 0,Y 202.154,Z 370.301,A -85,B 0,C 180,E1 -22896.481,E2 -22896.481} C_VEL
LIN {X 0,Y 200.505,Z 382.616,A -85,B 0,C 180,E1 -22897.298,E2 -22897.298} C_VEL
LIN {X 0,Y 198.776,Z 391.548,A -85,B 0,C 180,E1 -22898.19,E2 -22898.19} C_VEL
LIN {X 0,Y 196.562,Z 400.426,A -85,B 0,C 180,E1 -22899.359,E2 -22899.359} C_VEL
LIN {X 0,Y 194.082,Z 408.344,A -85,B 0,C 180,E1 -22900.667,E2 -22900.667} C_VEL
LIN {X 0,Y 191.311,Z 416.198,A -85,B 0,C 180,E1 -22902.337,E2 -22902.337} C_VEL
LIN {X 0,Y 188.489,Z 422.997,A -85,B 0,C 180,E1 -22904.131,E2 -22904.131} C_VEL
LIN {X 0,Y 185.397,Z 429.401,A -85,B 0,C 180,E1 -22906.224,E2 -22906.224} C_VEL
LIN {X 0,Y 181.889,Z 435.89,A -85,B 0,C 180,E1 -22908.939,E2 -22908.939} C_VEL
LIN {X 0,Y 178.757,Z 441.018,A -85,B 0,C 180,E1 -22911.828,E2 -22911.828} C_VEL
LIN {X 0,Y 176.154,Z 444.713,A -85,B 0,C 180,E1 -22914.655,E2 -22914.655} C_VEL
LIN {X 0,Y 173.554,Z 447.894,A -85,B 0,C 180,E1 -22918.236,E2 -22918.236} C_VEL
LIN {X 0,Y 172.121,Z 449.315,A -85,B 0,C 180,E1 -22920.661,E2 -22920.661} C_VEL
LIN {X 0,Y 170.964,Z 450.195,A -85,B 0,C 180,E1 -22923.116,E2 -22923.116} C_VEL
LIN {X 0,Y 170.099,Z 450.482,A -85,B 0,C 180,E1 -22925.596,E2 -22925.596} C_VEL
LIN {X 0,Y 169.434,Z 450.178,A -85,B 0,C 180,E1 -22928.08,E2 -22928.08} C_VEL
LIN {X 0,Y 169.042,Z 449.357,A -85,B 0,C 180,E1 -22930.574,E2 -22930.574} C_VEL
LIN {X 0,Y 168.902,Z 447.983,A -85,B 0,C 180,E1 -22933.109,E2 -22933.109} C_VEL
LIN {X 0,Y 169.049,Z 444.922,A -85,B 0,C 180,E1 -22936.783,E2 -22936.783} C_VEL
LIN {X 0,Y 169.393,Z 442.093,A -85,B 0,C 180,E1 -22939.24,E2 -22939.24} C_VEL
LIN {X 0,Y 170.137,Z 437.425,A -85,B 0,C 180,E1 -22942.403,E2 -22942.403} C_VEL
LIN {X 0,Y 171.002,Z 431.986,A -85,B 0,C 180,E1 -22945.286,E2 -22945.286} C_VEL
LIN {X 0,Y 172.207,Z 424.91,A -85,B 0,C 180,E1 -22948.246,E2 -22948.246} C_VEL
LIN {X 0,Y 173.633,Z 416.749,A -85,B 0,C 180,E1 -22950.87,E2 -22950.87} C_VEL
LIN {X 0,Y 174.952,Z 408.95,A -85,B 0,C 180,E1 -22952.879,E2 -22952.879} C_VEL
LIN {X 0,Y 176.232,Z 400.739,A -85,B 0,C 180,E1 -22954.575,E2 -22954.575} C_VEL
LIN {X 0,Y 177.395,Z 391.843,A -85,B 0,C 180,E1 -22956.026,E2 -22956.026} C_VEL
LIN {X 0,Y 178.311,Z 382.405,A -85,B 0,C 180,E1 -22957.207,E2 -22957.207} C_VEL
LIN {X 0,Y 179.23,Z 369.858,A -85,B 0,C 180,E1 -22958.259,E2 -22958.259} C_VEL
LIN {X 0,Y 179.98,Z 349.445,A -85,B 0,C 180,E1 -22959.15,E2 -22959.15} C_VEL
LIN {X 0,Y 180.854,Z 322.216,A -85,B 0,C 180,E1 -22960.212,E2 -22960.212} C_VEL
LIN {X 0,Y 176.568,Z 310.444,A -85,B 0,C 180,E1 -22961.264,E2 -22961.264} C_VEL
LIN {X 0,Y 171.748,Z 299.532,A -85,B 0,C 180,E1 -22962.414,E2 -22962.414} C_VEL
LIN {X 0,Y 171.632,Z 298.912,A -85,B 0,C 180,E1 -22962.475,E2 -22962.475} C_VEL
LIN {X 0,Y 171.52,Z 298.93,A -85,B 0,C 180,E1 -22966.668,E2 -22966.668} C_VEL
LIN {X 0,Y 171.513,Z 298.934,A -85,B 0,C 180,E1 -22969.56,E2 -22969.56} C_VEL
LIN {X 0,Y 171.418,Z 298.945,A -85,B 0,C 180,E1 -22975.602,E2 -22975.602} C_VEL
LIN {X 0,Y 171.393,Z 298.94,A -85,B 0,C 180,E1 -22980.577,E2 -22980.577} C_VEL
LIN {X 0,Y 171.37,Z 298.948,A -85,B 0,C 180,E1 -22985.041,E2 -22985.041} C_VEL
LIN {X 0,Y 171.322,Z 298.95,A -85,B 0,C 180,E1 -22988.807,E2 -22988.807} C_VEL
LIN {X 0,Y 171.3,Z 298.955,A -85,B 0,C 180,E1 -22994.225,E2 -22994.225} C_VEL
LIN {X 0,Y 171.318,Z 298.955,A -85,B 0,C 180,E1 -22998.988,E2 -22998.988} C_VEL
LIN {X 0,Y 171.372,Z 298.949,A -85,B 0,C 180,E1 -23002.048,E2 -23002.048} C_VEL
LIN {X 0,Y 171.384,Z 298.948,A -85,B 0,C 180,E1 -23005.1,E2 -23005.1} C_VEL
LIN {X 0,Y 171.398,Z 298.946,A -85,B 0,C 180,E1 -23010.535,E2 -23010.535} C_VEL
LIN {X 0,Y 171.44,Z 298.931,A -85,B 0,C 180,E1 -23015.808,E2 -23015.808} C_VEL
LIN {X 0,Y 172.126,Z 298.839,A -85,B 0,C 180,E1 -23023.401,E2 -23023.401} C_VEL
LIN {X 0,Y 173.583,Z 314.065,A -85,B 0,C 180,E1 -23024.525,E2 -23024.525} C_VEL
LIN {X 0,Y 172.666,Z 367.606,A -85,B 0,C 180,E1 -23028.817,E2 -23028.817} C_VEL
LIN {X 0,Y 172.382,Z 379.82,A -85,B 0,C 180,E1 -23030.167,E2 -23030.167} C_VEL
LIN {X 0,Y 171.906,Z 390.652,A -85,B 0,C 180,E1 -23031.781,E2 -23031.781} C_VEL
LIN {X 0,Y 171.502,Z 401.124,A -85,B 0,C 180,E1 -23033.833,E2 -23033.833} C_VEL
LIN {X 0,Y 171.141,Z 409.548,A -85,B 0,C 180,E1 -23035.887,E2 -23035.887} C_VEL
LIN {X 0,Y 170.9,Z 417.589,A -85,B 0,C 180,E1 -23038.24,E2 -23038.24} C_VEL
LIN {X 0,Y 170.475,Z 425.784,A -85,B 0,C 180,E1 -23041.189,E2 -23041.189} C_VEL
LIN {X 0,Y 170.542,Z 433.463,A -85,B 0,C 180,E1 -23044.735,E2 -23044.735} C_VEL
LIN {X 0,Y 170.893,Z 437.758,A -85,B 0,C 180,E1 -23047.094,E2 -23047.094} C_VEL
LIN {X 0,Y 171.851,Z 442.967,A -85,B 0,C 180,E1 -23050.612,E2 -23050.612} C_VEL
LIN {X 0,Y 173.571,Z 446.988,A -85,B 0,C 180,E1 -23054.068,E2 -23054.068} C_VEL
LIN {X 0,Y 175.378,Z 449.124,A -85,B 0,C 180,E1 -23056.298,E2 -23056.298} C_VEL
LIN {X 0,Y 177.284,Z 450.818,A -85,B 0,C 180,E1 -23058.497,E2 -23058.497} C_VEL
LIN {X 0,Y 179.792,Z 451.988,A -85,B 0,C 180,E1 -23060.605,E2 -23060.605} C_VEL
LIN {X 0,Y 185.525,Z 453.024,A -85,B 0,C 180,E1 -23064.633,E2 -23064.633} C_VEL
LIN {X 0,Y 188.871,Z 452.931,A -85,B 0,C 180,E1 -23066.528,E2 -23066.528} C_VEL
LIN {X 0,Y 192.509,Z 452.277,A -85,B 0,C 180,E1 -23068.34,E2 -23068.34} C_VEL
LIN {X 0,Y 196.368,Z 451.181,A -85,B 0,C 180,E1 -23070.077,E2 -23070.077} C_VEL
LIN {X 0,Y 200.513,Z 449.664,A -85,B 0,C 180,E1 -23071.725,E2 -23071.725} C_VEL
LIN {X 0,Y 207.096,Z 446.377,A -85,B 0,C 180,E1 -23074.058,E2 -23074.058} C_VEL
LIN {X 0,Y 214.107,Z 441.898,A -85,B 0,C 180,E1 -23076.223,E2 -23076.223} C_VEL
LIN {X 0,Y 221.581,Z 436.051,A -85,B 0,C 180,E1 -23078.212,E2 -23078.212} C_VEL
LIN {X 0,Y 229.409,Z 428.394,A -85,B 0,C 180,E1 -23080.047,E2 -23080.047} C_VEL
LIN {X 0,Y 234.795,Z 422.232,A -85,B 0,C 180,E1 -23081.192,E2 -23081.192} C_VEL
LIN {X 0,Y 241.772,Z 412.851,A -85,B 0,C 180,E1 -23082.525,E2 -23082.525} C_VEL
LIN {X 0,Y 247.8,Z 402.892,A -85,B 0,C 180,E1 -23083.599,E2 -23083.599} C_VEL
LIN {X 0,Y 250.909,Z 396.896,A -85,B 0,C 180,E1 -23084.114,E2 -23084.114} C_VEL
LIN {X 0,Y 251.428,Z 395.762,A -85,B 0,C 180,E1 -23084.337,E2 -23084.337} C_VEL
LIN {X 0,Y 250.962,Z 396.905,A -85,B 0,C 180,E1 -23085.147,E2 -23085.147} C_VEL
LIN {X 0,Y 244.818,Z 408.593,A -85,B 0,C 180,E1 -23085.964,E2 -23085.964} C_VEL
LIN {X 0,Y 238.823,Z 417.858,A -85,B 0,C 180,E1 -23086.827,E2 -23086.827} C_VEL
LIN {X 0,Y 237.059,Z 420.38,A -85,B 0,C 180,E1 -23087.107,E2 -23087.107} C_VEL
LIN {X 0,Y 233.537,Z 424.886,A -85,B 0,C 180,E1 -23087.521,E2 -23087.521} C_VEL
LIN {X 0,Y 226.755,Z 432.123,A -85,B 0,C 180,E1 -23087.863,E2 -23087.863} C_VEL
LIN {X 0,Y 219.601,Z 438.603,A -85,B 0,C 180,E1 -23088.337,E2 -23088.337} C_VEL
LIN {X 0,Y 215.539,Z 441.885,A -85,B 0,C 180,E1 -23088.968,E2 -23088.968} C_VEL
LIN {X 0,Y 206.785,Z 448.444,A -85,B 0,C 180,E1 -23091.041,E2 -23091.041} C_VEL
LIN {X 0,Y 199.287,Z 453,A -85,B 0,C 180,E1 -23093.164,E2 -23093.164} C_VEL
LIN {X 0,Y 194.558,Z 455.408,A -85,B 0,C 180,E1 -23094.692,E2 -23094.692} C_VEL
LIN {X 0,Y 190.11,Z 457.263,A -85,B 0,C 180,E1 -23096.322,E2 -23096.322} C_VEL
LIN {X 0,Y 185.939,Z 458.708,A -85,B 0,C 180,E1 -23098.051,E2 -23098.051} C_VEL
LIN {X 0,Y 182.089,Z 459.782,A -85,B 0,C 180,E1 -23099.883,E2 -23099.883} C_VEL
LIN {X 0,Y 178.593,Z 460.354,A -85,B 0,C 180,E1 -23101.821,E2 -23101.821} C_VEL
LIN {X 0,Y 172.445,Z 460.318,A -85,B 0,C 180,E1 -23105.948,E2 -23105.948} C_VEL
LIN {X 0,Y 170.056,Z 459.718,A -85,B 0,C 180,E1 -23108.164,E2 -23108.164} C_VEL
LIN {X 0,Y 166.606,Z 457.319,A -85,B 0,C 180,E1 -23112.825,E2 -23112.825} C_VEL
LIN {X 0,Y 165.032,Z 454.425,A -85,B 0,C 180,E1 -23116.454,E2 -23116.454} C_VEL
LIN {X 0,Y 164.423,Z 451.309,A -85,B 0,C 180,E1 -23119.568,E2 -23119.568} C_VEL
LIN {X 0,Y 162.68,Z 456.91,A -85,B 0,C 180,E1 -23123.393,E2 -23123.393} C_VEL
LIN {X 0,Y 162.256,Z 460.157,A -85,B 0,C 180,E1 -23126.33,E2 -23126.33} C_VEL
LIN {X 0,Y 162.299,Z 463.047,A -85,B 0,C 180,E1 -23130,E2 -23130} C_VEL
LIN {X 0,Y 161.998,Z 464.74,A -85,B 0,C 180,E1 -23133.697,E2 -23133.697} C_VEL
LIN {X 0,Y 162.175,Z 465.348,A -85,B 0,C 180,E1 -23137.47,E2 -23137.47} C_VEL
LIN {X 0,Y 162.618,Z 465.056,A -85,B 0,C 180,E1 -23139.954,E2 -23139.954} C_VEL
LIN {X 0,Y 163.342,Z 464.321,A -85,B 0,C 180,E1 -23142.423,E2 -23142.423} C_VEL
LIN {X 0,Y 164.384,Z 463.133,A -85,B 0,C 180,E1 -23144.863,E2 -23144.863} C_VEL
LIN {X 0,Y 166.508,Z 460.306,A -85,B 0,C 180,E1 -23148.455,E2 -23148.455} C_VEL
LIN {X 0,Y 169.372,Z 456.252,A -85,B 0,C 180,E1 -23151.928,E2 -23151.928} C_VEL
LIN {X 0,Y 172.974,Z 450.825,A -85,B 0,C 180,E1 -23155.253,E2 -23155.253} C_VEL
LIN {X 0,Y 176.384,Z 444.943,A -85,B 0,C 180,E1 -23157.916,E2 -23157.916} C_VEL
LIN {X 0,Y 180.157,Z 437.505,A -85,B 0,C 180,E1 -23160.473,E2 -23160.473} C_VEL
LIN {X 0,Y 183.572,Z 430.183,A -85,B 0,C 180,E1 -23162.41,E2 -23162.41} C_VEL
LIN {X 0,Y 186.61,Z 422.591,A -85,B 0,C 180,E1 -23164.013,E2 -23164.013} C_VEL
LIN {X 0,Y 189.406,Z 414.598,A -85,B 0,C 180,E1 -23165.336,E2 -23165.336} C_VEL
LIN {X 0,Y 192.083,Z 405.57,A -85,B 0,C 180,E1 -23166.481,E2 -23166.481} C_VEL
LIN {X 0,Y 194.705,Z 394.21,A -85,B 0,C 180,E1 -23167.525,E2 -23167.525} C_VEL
LIN {X 0,Y 196.31,Z 383.04,A -85,B 0,C 180,E1 -23168.184,E2 -23168.184} C_VEL
LIN {X 0,Y 197.314,Z 367.409,A -85,B 0,C 180,E1 -23168.808,E2 -23168.808} C_VEL
LIN {X 0,Y 196.04,Z 356.282,A -85,B 0,C 180,E1 -23169.769,E2 -23169.769} C_VEL
LIN {X 0,Y 191.149,Z 344.707,A -85,B 0,C 180,E1 -23171.984,E2 -23171.984} C_VEL
LIN {X 0,Y 186.375,Z 334.759,A -85,B 0,C 180,E1 -23174.299,E2 -23174.299} C_VEL
LIN {X 0,Y 180.721,Z 324.845,A -85,B 0,C 180,E1 -23177.248,E2 -23177.248} C_VEL
LIN {X 0,Y 177.019,Z 318.958,A -85,B 0,C 180,E1 -23179.365,E2 -23179.365} C_VEL
LIN {X 0,Y 173.484,Z 313.469,A -85,B 0,C 180,E1 -23181.578,E2 -23181.578} C_VEL
LIN {X 0,Y 170.204,Z 308.759,A -85,B 0,C 180,E1 -23183.857,E2 -23183.857} C_VEL
LIN {X 0,Y 169.261,Z 307.297,A -85,B 0,C 180,E1 -23184.57,E2 -23184.57} C_VEL
LIN {X 0,Y 165.009,Z 301.983,A -85,B 0,C 180,E1 -23188.022,E2 -23188.022} C_VEL
LIN {X 0,Y 164.52,Z 300.654,A -85,B 0,C 180,E1 -23188.689,E2 -23188.689} C_VEL
LIN {X 0,Y 164.386,Z 299.809,A -85,B 0,C 180,E1 -23189.837,E2 -23189.837} C_VEL
LIN {X 0,Y 164.404,Z 299.808,A -85,B 0,C 180,E1 -23194.684,E2 -23194.684} C_VEL
LIN {X 0,Y 164.491,Z 299.798,A -85,B 0,C 180,E1 -23200.045,E2 -23200.045} C_VEL
LIN {X 0,Y 164.504,Z 299.793,A -85,B 0,C 180,E1 -23205.14,E2 -23205.14} C_VEL
LIN {X 0,Y 164.771,Z 299.754,A -85,B 0,C 180,E1 -23210.169,E2 -23210.169} C_VEL
LIN {X 0,Y 164.832,Z 299.752,A -85,B 0,C 180,E1 -23212.643,E2 -23212.643} C_VEL
LIN {X 0,Y 165.043,Z 299.732,A -85,B 0,C 180,E1 -23217.552,E2 -23217.552} C_VEL
LIN {X 0,Y 165.291,Z 299.685,A -85,B 0,C 180,E1 -23219.992,E2 -23219.992} C_VEL
LIN {X 0,Y 164.752,Z 299.755,A -85,B 0,C 180,E1 -23224.886,E2 -23224.886} C_VEL
LIN {X 0,Y 164.823,Z 299.759,A -85,B 0,C 180,E1 -23227.341,E2 -23227.341} C_VEL
LIN {X 0,Y 164.698,Z 299.766,A -85,B 0,C 180,E1 -23231.053,E2 -23231.053} C_VEL
LIN {X 0,Y 164.488,Z 299.795,A -85,B 0,C 180,E1 -23235.004,E2 -23235.004} C_VEL
LIN {X 0,Y 165.205,Z 302.164,A -85,B 0,C 180,E1 -23235.806,E2 -23235.806} C_VEL
LIN {X 0,Y 167.135,Z 304.5,A -85,B 0,C 180,E1 -23237.425,E2 -23237.425} C_VEL
LIN {X 0,Y 169.038,Z 305.722,A -85,B 0,C 180,E1 -23238.806,E2 -23238.806} C_VEL
LIN {X 0,Y 170.766,Z 308.839,A -85,B 0,C 180,E1 -23240.153,E2 -23240.153} C_VEL
LIN {X 0,Y 173.243,Z 311.23,A -85,B 0,C 180,E1 -23241.784,E2 -23241.784} C_VEL
LIN {X 0,Y 175.628,Z 314.681,A -85,B 0,C 180,E1 -23243.306,E2 -23243.306} C_VEL
LIN {X 0,Y 177.102,Z 316.408,A -85,B 0,C 180,E1 -23244.165,E2 -23244.165} C_VEL
LIN {X 0,Y 180.844,Z 321.541,A -85,B 0,C 180,E1 -23246.255,E2 -23246.255} C_VEL
LIN {X 0,Y 185.77,Z 328.526,A -85,B 0,C 180,E1 -23248.752,E2 -23248.752} C_VEL
LIN {X 0,Y 192.93,Z 340.124,A -85,B 0,C 180,E1 -23252.029,E2 -23252.029} C_VEL
LIN {X 0,Y 198.372,Z 350.279,A -85,B 0,C 180,E1 -23254.291,E2 -23254.291} C_VEL
LIN {X 0,Y 197.069,Z 370.217,A -85,B 0,C 180,E1 -23255.053,E2 -23255.053} C_VEL
LIN {X 0,Y 195.52,Z 381.961,A -85,B 0,C 180,E1 -23255.812,E2 -23255.812} C_VEL
LIN {X 0,Y 193.33,Z 392.625,A -85,B 0,C 180,E1 -23256.894,E2 -23256.894} C_VEL
LIN {X 0,Y 190.938,Z 401.606,A -85,B 0,C 180,E1 -23258.116,E2 -23258.116} C_VEL
LIN {X 0,Y 188.158,Z 409.956,A -85,B 0,C 180,E1 -23259.561,E2 -23259.561} C_VEL
LIN {X 0,Y 184.601,Z 419.219,A -85,B 0,C 180,E1 -23261.657,E2 -23261.657} C_VEL
LIN {X 0,Y 180.969,Z 426.96,A -85,B 0,C 180,E1 -23263.96,E2 -23263.96} C_VEL
LIN {X 0,Y 177.75,Z 432.876,A -85,B 0,C 180,E1 -23266.218,E2 -23266.218} C_VEL
LIN {X 0,Y 174.914,Z 437.59,A -85,B 0,C 180,E1 -23268.474,E2 -23268.474} C_VEL
LIN {X 0,Y 172.452,Z 441.362,A -85,B 0,C 180,E1 -23270.728,E2 -23270.728} C_VEL
LIN {X 0,Y 170.078,Z 444.584,A -85,B 0,C 180,E1 -23273.19,E2 -23273.19} C_VEL
LIN {X 0,Y 167.217,Z 447.924,A -85,B 0,C 180,E1 -23276.881,E2 -23276.881} C_VEL
LIN {X 0,Y 165.647,Z 449.47,A -85,B 0,C 180,E1 -23279.395,E2 -23279.395} C_VEL
LIN {X 0,Y 164.325,Z 450.425,A -85,B 0,C 180,E1 -23281.937,E2 -23281.937} C_VEL
LIN {X 0,Y 163.274,Z 450.78,A -85,B 0,C 180,E1 -23284.656,E2 -23284.656} C_VEL
LIN {X 0,Y 162.549,Z 450.58,A -85,B 0,C 180,E1 -23287.1,E2 -23287.1} C_VEL
LIN {X 0,Y 162.056,Z 449.881,A -85,B 0,C 180,E1 -23289.7,E2 -23289.7} C_VEL
LIN {X 0,Y 161.813,Z 448.321,A -85,B 0,C 180,E1 -23292.814,E2 -23292.814} C_VEL
LIN {X 0,Y 161.915,Z 445.692,A -85,B 0,C 180,E1 -23296.189,E2 -23296.189} C_VEL
LIN {X 0,Y 162.223,Z 442.997,A -85,B 0,C 180,E1 -23298.758,E2 -23298.758} C_VEL
LIN {X 0,Y 163.073,Z 437.678,A -85,B 0,C 180,E1 -23302.572,E2 -23302.572} C_VEL
LIN {X 0,Y 164.027,Z 431.983,A -85,B 0,C 180,E1 -23305.7,E2 -23305.7} C_VEL
LIN {X 0,Y 165.293,Z 424.778,A -85,B 0,C 180,E1 -23308.782,E2 -23308.782} C_VEL
LIN {X 0,Y 166.773,Z 416.514,A -85,B 0,C 180,E1 -23311.51,E2 -23311.51} C_VEL
LIN {X 0,Y 168.199,Z 408.59,A -85,B 0,C 180,E1 -23313.594,E2 -23313.594} C_VEL
LIN {X 0,Y 169.425,Z 400.878,A -85,B 0,C 180,E1 -23315.23,E2 -23315.23} C_VEL
LIN {X 0,Y 170.759,Z 391.133,A -85,B 0,C 180,E1 -23316.855,E2 -23316.855} C_VEL
LIN {X 0,Y 171.922,Z 379.062,A -85,B 0,C 180,E1 -23318.304,E2 -23318.304} C_VEL
LIN {X 0,Y 172.581,Z 369.201,A -85,B 0,C 180,E1 -23319.066,E2 -23319.066} C_VEL
LIN {X 0,Y 173.649,Z 341.714,A -85,B 0,C 180,E1 -23320.253,E2 -23320.253} C_VEL
LIN {X 0,Y 174.148,Z 323.569,A -85,B 0,C 180,E1 -23320.999,E2 -23320.999} C_VEL
LIN {X 0,Y 170.624,Z 313.79,A -85,B 0,C 180,E1 -23321.92,E2 -23321.92} C_VEL
LIN {X 0,Y 164.631,Z 300.417,A -85,B 0,C 180,E1 -23323.434,E2 -23323.434} C_VEL
LIN {X 0,Y 164.541,Z 299.799,A -85,B 0,C 180,E1 -23323.541,E2 -23323.541} C_VEL
LIN {X 0,Y 164.452,Z 299.814,A -85,B 0,C 180,E1 -23327.407,E2 -23327.407} C_VEL
LIN {X 0,Y 164.447,Z 299.813,A -85,B 0,C 180,E1 -23329.993,E2 -23329.993} C_VEL
LIN {X 0,Y 164.345,Z 299.825,A -85,B 0,C 180,E1 -23336.121,E2 -23336.121} C_VEL
LIN {X 0,Y 164.329,Z 299.816,A -85,B 0,C 180,E1 -23341.22,E2 -23341.22} C_VEL
LIN {X 0,Y 164.258,Z 299.834,A -85,B 0,C 180,E1 -23346.8,E2 -23346.8} C_VEL
LIN {X 0,Y 164.266,Z 299.834,A -85,B 0,C 180,E1 -23349.924,E2 -23349.924} C_VEL
LIN {X 0,Y 164.261,Z 299.833,A -85,B 0,C 180,E1 -23353.349,E2 -23353.349} C_VEL
LIN {X 0,Y 164.245,Z 299.837,A -85,B 0,C 180,E1 -23356.806,E2 -23356.806} C_VEL
LIN {X 0,Y 164.279,Z 299.828,A -85,B 0,C 180,E1 -23360.36,E2 -23360.36} C_VEL
LIN {X 0,Y 164.316,Z 299.829,A -85,B 0,C 180,E1 -23364.357,E2 -23364.357} C_VEL
LIN {X 0,Y 164.359,Z 299.82,A -85,B 0,C 180,E1 -23369.138,E2 -23369.138} C_VEL
LIN {X 0,Y 164.387,Z 299.813,A -85,B 0,C 180,E1 -23374.699,E2 -23374.699} C_VEL
LIN {X 0,Y 164.909,Z 299.734,A -85,B 0,C 180,E1 -23382.652,E2 -23382.652} C_VEL
LIN {X 0,Y 165.169,Z 299.806,A -85,B 0,C 180,E1 -23383.794,E2 -23383.794} C_VEL
LIN {X 0,Y 166.565,Z 314.124,A -85,B 0,C 180,E1 -23384.875,E2 -23384.875} C_VEL
LIN {X 0,Y 165.834,Z 366.029,A -85,B 0,C 180,E1 -23389.258,E2 -23389.258} C_VEL
LIN {X 0,Y 165.529,Z 378.825,A -85,B 0,C 180,E1 -23390.693,E2 -23390.693} C_VEL
LIN {X 0,Y 165.101,Z 389.657,A -85,B 0,C 180,E1 -23392.364,E2 -23392.364} C_VEL
LIN {X 0,Y 164.686,Z 400.466,A -85,B 0,C 180,E1 -23394.498,E2 -23394.498} C_VEL
LIN {X 0,Y 164.29,Z 410.093,A -85,B 0,C 180,E1 -23396.943,E2 -23396.943} C_VEL
LIN {X 0,Y 164.045,Z 417.967,A -85,B 0,C 180,E1 -23399.394,E2 -23399.394} C_VEL
LIN {X 0,Y 163.694,Z 425.969,A -85,B 0,C 180,E1 -23402.468,E2 -23402.468} C_VEL
LIN {X 0,Y 163.904,Z 433.688,A -85,B 0,C 180,E1 -23406.161,E2 -23406.161} C_VEL
LIN {X 0,Y 164.364,Z 437.953,A -85,B 0,C 180,E1 -23408.615,E2 -23408.615} C_VEL
LIN {X 0,Y 165.787,Z 443.831,A -85,B 0,C 180,E1 -23412.834,E2 -23412.834} C_VEL
LIN {X 0,Y 167.653,Z 447.224,A -85,B 0,C 180,E1 -23415.819,E2 -23415.819} C_VEL
LIN {X 0,Y 170.598,Z 450.254,A -85,B 0,C 180,E1 -23419.25,E2 -23419.25} C_VEL
LIN {X 0,Y 175.986,Z 452.836,A -85,B 0,C 180,E1 -23423.545,E2 -23423.545} C_VEL
LIN {X 0,Y 180.015,Z 453.522,A -85,B 0,C 180,E1 -23426.109,E2 -23426.109} C_VEL
LIN {X 0,Y 186.347,Z 453.244,A -85,B 0,C 180,E1 -23429.366,E2 -23429.366} C_VEL
LIN {X 0,Y 190.343,Z 452.556,A -85,B 0,C 180,E1 -23431.132,E2 -23431.132} C_VEL
LIN {X 0,Y 194.625,Z 451.292,A -85,B 0,C 180,E1 -23432.803,E2 -23432.803} C_VEL
LIN {X 0,Y 201.442,Z 448.608,A -85,B 0,C 180,E1 -23435.152,E2 -23435.152} C_VEL
LIN {X 0,Y 208.694,Z 444.74,A -85,B 0,C 180,E1 -23437.319,E2 -23437.319} C_VEL
LIN {X 0,Y 216.333,Z 439.5,A -85,B 0,C 180,E1 -23439.315,E2 -23439.315} C_VEL
LIN {X 0,Y 222.632,Z 434.383,A -85,B 0,C 180,E1 -23440.744,E2 -23440.744} C_VEL
LIN {X 0,Y 229.961,Z 427.299,A -85,B 0,C 180,E1 -23442.255,E2 -23442.255} C_VEL
LIN {X 0,Y 237.107,Z 419.12,A -85,B 0,C 180,E1 -23443.568,E2 -23443.568} C_VEL
LIN {X 0,Y 241.489,Z 413.206,A -85,B 0,C 180,E1 -23444.309,E2 -23444.309} C_VEL
LIN {X 0,Y 240.157,Z 415.094,A -85,B 0,C 180,E1 -23444.783,E2 -23444.783} C_VEL
LIN {X 0,Y 233.878,Z 423.451,A -85,B 0,C 180,E1 -23445.68,E2 -23445.68} C_VEL
LIN {X 0,Y 227.762,Z 430.429,A -85,B 0,C 180,E1 -23446.641,E2 -23446.641} C_VEL
LIN {X 0,Y 218.99,Z 439.017,A -85,B 0,C 180,E1 -23448.246,E2 -23448.246} C_VEL
LIN {X 0,Y 215.539,Z 441.885,A -85,B 0,C 180,E1 -23448.968,E2 -23448.968} C_VEL
LIN {X 0,Y 211.317,Z 445.086,A -85,B 0,C 180,E1 -23449.693,E2 -23449.693} C_VEL
LIN {X 0,Y 203.298,Z 449.874,A -85,B 0,C 180,E1 -23450.624,E2 -23450.624} C_VEL
LIN {X 0,Y 195.167,Z 453.789,A -85,B 0,C 180,E1 -23451.751,E2 -23451.751} C_VEL
LIN {X 0,Y 190.832,Z 455.535,A -85,B 0,C 180,E1 -23452.796,E2 -23452.796} C_VEL
LIN {X 0,Y 184.248,Z 457.867,A -85,B 0,C 180,E1 -23455.098,E2 -23455.098} C_VEL
LIN {X 0,Y 179.958,Z 459.02,A -85,B 0,C 180,E1 -23456.855,E2 -23456.855} C_VEL
LIN {X 0,Y 172.392,Z 459.977,A -85,B 0,C 180,E1 -23460.711,E2 -23460.711} C_VEL
LIN {X 0,Y 169.077,Z 459.932,A -85,B 0,C 180,E1 -23462.791,E2 -23462.791} C_VEL
LIN {X 0,Y 166.047,Z 459.357,A -85,B 0,C 180,E1 -23464.959,E2 -23464.959} C_VEL
LIN {X 0,Y 161.598,Z 457.324,A -85,B 0,C 180,E1 -23469.639,E2 -23469.639} C_VEL
LIN {X 0,Y 158.855,Z 453.569,A -85,B 0,C 180,E1 -23474.606,E2 -23474.606} C_VEL
LIN {X 0,Y 157.887,Z 449.559,A -85,B 0,C 180,E1 -23478.607,E2 -23478.607} C_VEL
LIN {X 0,Y 155.908,Z 455.189,A -85,B 0,C 180,E1 -23482.227,E2 -23482.227} C_VEL
LIN {X 0,Y 155.31,Z 458.233,A -85,B 0,C 180,E1 -23484.807,E2 -23484.807} C_VEL
LIN {X 0,Y 155.154,Z 460.658,A -85,B 0,C 180,E1 -23487.403,E2 -23487.403} C_VEL
LIN {X 0,Y 155.236,Z 462.534,A -85,B 0,C 180,E1 -23489.999,E2 -23489.999} C_VEL
LIN {X 0,Y 154.94,Z 464.212,A -85,B 0,C 180,E1 -23493.607,E2 -23493.607} C_VEL
LIN {X 0,Y 154.94,Z 464.716,A -85,B 0,C 180,E1 -23495.204,E2 -23495.204} C_VEL
LIN {X 0,Y 155.147,Z 464.983,A -85,B 0,C 180,E1 -23497.81,E2 -23497.81} C_VEL
LIN {X 0,Y 155.624,Z 464.764,A -85,B 0,C 180,E1 -23500.407,E2 -23500.407} C_VEL
LIN {X 0,Y 156.4,Z 464.103,A -85,B 0,C 180,E1 -23502.984,E2 -23502.984} C_VEL
LIN {X 0,Y 157.528,Z 462.992,A -85,B 0,C 180,E1 -23505.526,E2 -23505.526} C_VEL
LIN {X 0,Y 159.786,Z 460.244,A -85,B 0,C 180,E1 -23509.261,E2 -23509.261} C_VEL
LIN {X 0,Y 162.809,Z 456.275,A -85,B 0,C 180,E1 -23512.861,E2 -23512.861} C_VEL
LIN {X 0,Y 165.266,Z 452.868,A -85,B 0,C 180,E1 -23515.166,E2 -23515.166} C_VEL
LIN {X 0,Y 168.676,Z 447.592,A -85,B 0,C 180,E1 -23517.952,E2 -23517.952} C_VEL
LIN {X 0,Y 171.752,Z 442.437,A -85,B 0,C 180,E1 -23520.083,E2 -23520.083} C_VEL
LIN {X 0,Y 174.109,Z 437.961,A -85,B 0,C 180,E1 -23521.651,E2 -23521.651} C_VEL
LIN {X 0,Y 177.658,Z 430.796,A -85,B 0,C 180,E1 -23523.63,E2 -23523.63} C_VEL
LIN {X 0,Y 180.804,Z 423.396,A -85,B 0,C 180,E1 -23525.264,E2 -23525.264} C_VEL
LIN {X 0,Y 183.846,Z 415.202,A -85,B 0,C 180,E1 -23526.677,E2 -23526.677} C_VEL
LIN {X 0,Y 186.436,Z 406.968,A -85,B 0,C 180,E1 -23527.775,E2 -23527.775} C_VEL
LIN {X 0,Y 188.633,Z 398.605,A -85,B 0,C 180,E1 -23528.613,E2 -23528.613} C_VEL
LIN {X 0,Y 190.374,Z 389.352,A -85,B 0,C 180,E1 -23529.326,E2 -23529.326} C_VEL
LIN {X 0,Y 191.508,Z 380.76,A -85,B 0,C 180,E1 -23529.772,E2 -23529.772} C_VEL
LIN {X 0,Y 192.303,Z 368.356,A -85,B 0,C 180,E1 -23530.274,E2 -23530.274} C_VEL
LIN {X 0,Y 191.273,Z 359.209,A -85,B 0,C 180,E1 -23531.119,E2 -23531.119} C_VEL
LIN {X 0,Y 186.198,Z 346.92,A -85,B 0,C 180,E1 -23533.621,E2 -23533.621} C_VEL
LIN {X 0,Y 181.59,Z 337.641,A -85,B 0,C 180,E1 -23536.022,E2 -23536.022} C_VEL
LIN {X 0,Y 177.097,Z 329.623,A -85,B 0,C 180,E1 -23538.555,E2 -23538.555} C_VEL
LIN {X 0,Y 173.78,Z 324.171,A -85,B 0,C 180,E1 -23540.59,E2 -23540.59} C_VEL
LIN {X 0,Y 170.699,Z 319.201,A -85,B 0,C 180,E1 -23542.668,E2 -23542.668} C_VEL
LIN {X 0,Y 167.466,Z 314.178,A -85,B 0,C 180,E1 -23545.105,E2 -23545.105} C_VEL
LIN {X 0,Y 162.832,Z 308.029,A -85,B 0,C 180,E1 -23549.083,E2 -23549.083} C_VEL
LIN {X 0,Y 161.932,Z 306.519,A -85,B 0,C 180,E1 -23549.997,E2 -23549.997} C_VEL
LIN {X 0,Y 159.129,Z 304.656,A -85,B 0,C 180,E1 -23552.8,E2 -23552.8} C_VEL
LIN {X 0,Y 157.754,Z 302.284,A -85,B 0,C 180,E1 -23554.601,E2 -23554.601} C_VEL
LIN {X 0,Y 157.339,Z 300.693,A -85,B 0,C 180,E1 -23555.412,E2 -23555.412} C_VEL
LIN {X 0,Y 157.398,Z 300.678,A -85,B 0,C 180,E1 -23559.664,E2 -23559.664} C_VEL
LIN {X 0,Y 157.441,Z 300.668,A -85,B 0,C 180,E1 -23564.457,E2 -23564.457} C_VEL
LIN {X 0,Y 157.693,Z 300.633,A -85,B 0,C 180,E1 -23569.723,E2 -23569.723} C_VEL
LIN {X 0,Y 157.769,Z 300.635,A -85,B 0,C 180,E1 -23572.312,E2 -23572.312} C_VEL
LIN {X 0,Y 158.253,Z 300.562,A -85,B 0,C 180,E1 -23579.992,E2 -23579.992} C_VEL
LIN {X 0,Y 157.76,Z 300.642,A -85,B 0,C 180,E1 -23587.672,E2 -23587.672} C_VEL
LIN {X 0,Y 157.724,Z 300.695,A -85,B 0,C 180,E1 -23588.802,E2 -23588.802} C_VEL
LIN {X 0,Y 158.408,Z 302.939,A -85,B 0,C 180,E1 -23589.891,E2 -23589.891} C_VEL
LIN {X 0,Y 160.37,Z 305.473,A -85,B 0,C 180,E1 -23592.163,E2 -23592.163} C_VEL
LIN {X 0,Y 162.401,Z 306.695,A -85,B 0,C 180,E1 -23594.08,E2 -23594.08} C_VEL
LIN {X 0,Y 163.851,Z 309.537,A -85,B 0,C 180,E1 -23595.541,E2 -23595.541} C_VEL
LIN {X 0,Y 166.214,Z 311.761,A -85,B 0,C 180,E1 -23597.485,E2 -23597.485} C_VEL
LIN {X 0,Y 166.915,Z 312.471,A -85,B 0,C 180,E1 -23598.031,E2 -23598.031} C_VEL
LIN {X 0,Y 169.111,Z 315.805,A -85,B 0,C 180,E1 -23599.754,E2 -23599.754} C_VEL
LIN {X 0,Y 170.857,Z 317.625,A -85,B 0,C 180,E1 -23600.958,E2 -23600.958} C_VEL
LIN {X 0,Y 173.67,Z 321.388,A -85,B 0,C 180,E1 -23602.816,E2 -23602.816} C_VEL
LIN {X 0,Y 178.259,Z 327.892,A -85,B 0,C 180,E1 -23605.535,E2 -23605.535} C_VEL
LIN {X 0,Y 182.977,Z 334.867,A -85,B 0,C 180,E1 -23608.042,E2 -23608.042} C_VEL
LIN {X 0,Y 189.122,Z 345.046,A -85,B 0,C 180,E1 -23611,E2 -23611} C_VEL
LIN {X 0,Y 193.362,Z 353.058,A -85,B 0,C 180,E1 -23612.893,E2 -23612.893} C_VEL
LIN {X 0,Y 191.964,Z 372.041,A -85,B 0,C 180,E1 -23613.637,E2 -23613.637} C_VEL
LIN {X 0,Y 190.139,Z 383.955,A -85,B 0,C 180,E1 -23614.489,E2 -23614.489} C_VEL
LIN {X 0,Y 188.419,Z 392.072,A -85,B 0,C 180,E1 -23615.321,E2 -23615.321} C_VEL
LIN {X 0,Y 185.931,Z 401.22,A -85,B 0,C 180,E1 -23616.561,E2 -23616.561} C_VEL
LIN {X 0,Y 183.372,Z 408.678,A -85,B 0,C 180,E1 -23617.812,E2 -23617.812} C_VEL
LIN {X 0,Y 180.619,Z 415.838,A -85,B 0,C 180,E1 -23619.345,E2 -23619.345} C_VEL
LIN {X 0,Y 177.504,Z 422.836,A -85,B 0,C 180,E1 -23621.213,E2 -23621.213} C_VEL
LIN {X 0,Y 174.033,Z 429.378,A -85,B 0,C 180,E1 -23623.374,E2 -23623.374} C_VEL
LIN {X 0,Y 170.86,Z 434.759,A -85,B 0,C 180,E1 -23625.633,E2 -23625.633} C_VEL
LIN {X 0,Y 167.948,Z 439.184,A -85,B 0,C 180,E1 -23627.969,E2 -23627.969} C_VEL
LIN {X 0,Y 165.34,Z 442.797,A -85,B 0,C 180,E1 -23630.388,E2 -23630.388} C_VEL
LIN {X 0,Y 161.936,Z 446.881,A -85,B 0,C 180,E1 -23634.134,E2 -23634.134} C_VEL
LIN {X 0,Y 159.247,Z 449.589,A -85,B 0,C 180,E1 -23638.023,E2 -23638.023} C_VEL
LIN {X 0,Y 157.759,Z 450.59,A -85,B 0,C 180,E1 -23640.657,E2 -23640.657} C_VEL
LIN {X 0,Y 156.345,Z 451.117,A -85,B 0,C 180,E1 -23644.009,E2 -23644.009} C_VEL
LIN {X 0,Y 155.111,Z 450.404,A -85,B 0,C 180,E1 -23648.748,E2 -23648.748} C_VEL
LIN {X 0,Y 154.72,Z 448.653,A -85,B 0,C 180,E1 -23652.501,E2 -23652.501} C_VEL
LIN {X 0,Y 154.76,Z 446.466,A -85,B 0,C 180,E1 -23655.537,E2 -23655.537} C_VEL
LIN {X 0,Y 155.233,Z 442.326,A -85,B 0,C 180,E1 -23659.567,E2 -23659.567} C_VEL
LIN {X 0,Y 155.925,Z 438.332,A -85,B 0,C 180,E1 -23662.489,E2 -23662.489} C_VEL
LIN {X 0,Y 156.818,Z 433.187,A -85,B 0,C 180,E1 -23665.502,E2 -23665.502} C_VEL
LIN {X 0,Y 158.055,Z 426.28,A -85,B 0,C 180,E1 -23668.727,E2 -23668.727} C_VEL
LIN {X 0,Y 159.768,Z 417.313,A -85,B 0,C 180,E1 -23671.891,E2 -23671.891} C_VEL
LIN {X 0,Y 161.241,Z 409.483,A -85,B 0,C 180,E1 -23674.062,E2 -23674.062} C_VEL
LIN {X 0,Y 162.51,Z 401.957,A -85,B 0,C 180,E1 -23675.752,E2 -23675.752} C_VEL
LIN {X 0,Y 163.665,Z 393.992,A -85,B 0,C 180,E1 -23677.19,E2 -23677.19} C_VEL
LIN {X 0,Y 164.642,Z 385.186,A -85,B 0,C 180,E1 -23678.438,E2 -23678.438} C_VEL
LIN {X 0,Y 165.508,Z 375.945,A -85,B 0,C 180,E1 -23679.394,E2 -23679.394} C_VEL
LIN {X 0,Y 166.044,Z 366.571,A -85,B 0,C 180,E1 -23680.053,E2 -23680.053} C_VEL
LIN {X 0,Y 167.605,Z 325.137,A -85,B 0,C 180,E1 -23681.82,E2 -23681.82} C_VEL
LIN {X 0,Y 163.066,Z 313.211,A -85,B 0,C 180,E1 -23683.06,E2 -23683.06} C_VEL
LIN {X 0,Y 157.583,Z 301.393,A -85,B 0,C 180,E1 -23684.538,E2 -23684.538} C_VEL
LIN {X 0,Y 157.442,Z 300.687,A -85,B 0,C 180,E1 -23684.626,E2 -23684.626} C_VEL
LIN {X 0,Y 157.366,Z 300.694,A -85,B 0,C 180,E1 -23690.334,E2 -23690.334} C_VEL
LIN {X 0,Y 157.286,Z 300.704,A -85,B 0,C 180,E1 -23696.686,E2 -23696.686} C_VEL
LIN {X 0,Y 157.241,Z 300.699,A -85,B 0,C 180,E1 -23702.436,E2 -23702.436} C_VEL
LIN {X 0,Y 157.237,Z 300.708,A -85,B 0,C 180,E1 -23706.45,E2 -23706.45} C_VEL
LIN {X 0,Y 157.171,Z 300.717,A -85,B 0,C 180,E1 -23712.125,E2 -23712.125} C_VEL
LIN {X 0,Y 157.175,Z 300.719,A -85,B 0,C 180,E1 -23717.891,E2 -23717.891} C_VEL
LIN {X 0,Y 157.254,Z 300.709,A -85,B 0,C 180,E1 -23723.559,E2 -23723.559} C_VEL
LIN {X 0,Y 157.271,Z 300.702,A -85,B 0,C 180,E1 -23728.11,E2 -23728.11} C_VEL
LIN {X 0,Y 157.3,Z 300.702,A -85,B 0,C 180,E1 -23733.472,E2 -23733.472} C_VEL
LIN {X 0,Y 157.494,Z 300.649,A -85,B 0,C 180,E1 -23739.572,E2 -23739.572} C_VEL
LIN {X 0,Y 158.185,Z 300.612,A -85,B 0,C 180,E1 -23744.218,E2 -23744.218} C_VEL
LIN {X 0,Y 159.561,Z 314.173,A -85,B 0,C 180,E1 -23745.297,E2 -23745.297} C_VEL
LIN {X 0,Y 158.933,Z 368.071,A -85,B 0,C 180,E1 -23750.142,E2 -23750.142} C_VEL
LIN {X 0,Y 158.675,Z 379.799,A -85,B 0,C 180,E1 -23751.572,E2 -23751.572} C_VEL
LIN {X 0,Y 158.241,Z 390.439,A -85,B 0,C 180,E1 -23753.313,E2 -23753.313} C_VEL
LIN {X 0,Y 157.875,Z 400.988,A -85,B 0,C 180,E1 -23755.54,E2 -23755.54} C_VEL
LIN {X 0,Y 157.54,Z 410.385,A -85,B 0,C 180,E1 -23758.091,E2 -23758.091} C_VEL
LIN {X 0,Y 157.352,Z 416.355,A -85,B 0,C 180,E1 -23760.008,E2 -23760.008} C_VEL
LIN {X 0,Y 157.001,Z 424.605,A -85,B 0,C 180,E1 -23763.216,E2 -23763.216} C_VEL
LIN {X 0,Y 157.244,Z 432.63,A -85,B 0,C 180,E1 -23767.068,E2 -23767.068} C_VEL
LIN {X 0,Y 157.874,Z 438.011,A -85,B 0,C 180,E1 -23770.265,E2 -23770.265} C_VEL
LIN {X 0,Y 159.296,Z 443.083,A -85,B 0,C 180,E1 -23773.921,E2 -23773.921} C_VEL
LIN {X 0,Y 161.926,Z 447.37,A -85,B 0,C 180,E1 -23777.695,E2 -23777.695} C_VEL
LIN {X 0,Y 163.954,Z 449.616,A -85,B 0,C 180,E1 -23780.063,E2 -23780.063} C_VEL
LIN {X 0,Y 166.624,Z 451.369,A -85,B 0,C 180,E1 -23782.317,E2 -23782.317} C_VEL
LIN {X 0,Y 172.747,Z 453.533,A -85,B 0,C 180,E1 -23786.592,E2 -23786.592} C_VEL
LIN {X 0,Y 176.314,Z 454.049,A -85,B 0,C 180,E1 -23788.584,E2 -23788.584} C_VEL
LIN {X 0,Y 180.214,Z 454.019,A -85,B 0,C 180,E1 -23790.47,E2 -23790.47} C_VEL
LIN {X 0,Y 184.35,Z 453.573,A -85,B 0,C 180,E1 -23792.264,E2 -23792.264} C_VEL
LIN {X 0,Y 188.772,Z 452.735,A -85,B 0,C 180,E1 -23793.956,E2 -23793.956} C_VEL
LIN {X 0,Y 193.418,Z 451.442,A -85,B 0,C 180,E1 -23795.554,E2 -23795.554} C_VEL
LIN {X 0,Y 200.77,Z 448.501,A -85,B 0,C 180,E1 -23797.784,E2 -23797.784} C_VEL
LIN {X 0,Y 208.507,Z 444.403,A -85,B 0,C 180,E1 -23799.829,E2 -23799.829} C_VEL
LIN {X 0,Y 215.959,Z 439.45,A -85,B 0,C 180,E1 -23801.539,E2 -23801.539} C_VEL
LIN {X 0,Y 223.592,Z 433.421,A -85,B 0,C 180,E1 -23803.066,E2 -23803.066} C_VEL
LIN {X 0,Y 228.078,Z 429.247,A -85,B 0,C 180,E1 -23803.899,E2 -23803.899} C_VEL
LIN {X 0,Y 228.985,Z 428.411,A -85,B 0,C 180,E1 -23804.473,E2 -23804.473} C_VEL
LIN {X 0,Y 221.283,Z 435.914,A -85,B 0,C 180,E1 -23805.675,E2 -23805.675} C_VEL
LIN {X 0,Y 213.835,Z 442.065,A -85,B 0,C 180,E1 -23807.001,E2 -23807.001} C_VEL
LIN {X 0,Y 204.057,Z 448.788,A -85,B 0,C 180,E1 -23809.126,E2 -23809.126} C_VEL
LIN {X 0,Y 196.195,Z 453.072,A -85,B 0,C 180,E1 -23811.179,E2 -23811.179} C_VEL
LIN {X 0,Y 190.832,Z 455.535,A -85,B 0,C 180,E1 -23812.796,E2 -23812.796} C_VEL
LIN {X 0,Y 187.736,Z 456.589,A -85,B 0,C 180,E1 -23813.513,E2 -23813.513} C_VEL
LIN {X 0,Y 181.629,Z 457.966,A -85,B 0,C 180,E1 -23814.338,E2 -23814.338} C_VEL
LIN {X 0,Y 175.646,Z 458.883,A -85,B 0,C 180,E1 -23815.27,E2 -23815.27} C_VEL
LIN {X 0,Y 172.785,Z 459.125,A -85,B 0,C 180,E1 -23816.161,E2 -23816.161} C_VEL
LIN {X 0,Y 169.998,Z 459.437,A -85,B 0,C 180,E1 -23817.49,E2 -23817.49} C_VEL
LIN {X 0,Y 166.264,Z 459.42,A -85,B 0,C 180,E1 -23819.519,E2 -23819.519} C_VEL
LIN {X 0,Y 159.742,Z 458.272,A -85,B 0,C 180,E1 -23823.898,E2 -23823.898} C_VEL
LIN {X 0,Y 157.177,Z 457.129,A -85,B 0,C 180,E1 -23826.27,E2 -23826.27} C_VEL
LIN {X 0,Y 153.519,Z 453.773,A -85,B 0,C 180,E1 -23831.309,E2 -23831.309} C_VEL
LIN {X 0,Y 151.925,Z 450.141,A -85,B 0,C 180,E1 -23835.26,E2 -23835.26} C_VEL
LIN {X 0,Y 151.43,Z 447.758,A -85,B 0,C 180,E1 -23837.557,E2 -23837.557} C_VEL
LIN {X 0,Y 150.169,Z 450.658,A -85,B 0,C 180,E1 -23839.21,E2 -23839.21} C_VEL
LIN {X 0,Y 148.529,Z 456.046,A -85,B 0,C 180,E1 -23843.206,E2 -23843.206} C_VEL
LIN {X 0,Y 148.089,Z 460.065,A -85,B 0,C 180,E1 -23847.279,E2 -23847.279} C_VEL
LIN {X 0,Y 148.173,Z 462.02,A -85,B 0,C 180,E1 -23849.999,E2 -23849.999} C_VEL
LIN {X 0,Y 147.877,Z 463.674,A -85,B 0,C 180,E1 -23853.476,E2 -23853.476} C_VEL
LIN {X 0,Y 147.865,Z 464.31,A -85,B 0,C 180,E1 -23855.454,E2 -23855.454} C_VEL
LIN {X 0,Y 148.095,Z 464.617,A -85,B 0,C 180,E1 -23858.184,E2 -23858.184} C_VEL
LIN {X 0,Y 148.626,Z 464.472,A -85,B 0,C 180,E1 -23860.902,E2 -23860.902} C_VEL
LIN {X 0,Y 149.483,Z 463.887,A -85,B 0,C 180,E1 -23863.596,E2 -23863.596} C_VEL
LIN {X 0,Y 150.68,Z 462.833,A -85,B 0,C 180,E1 -23866.251,E2 -23866.251} C_VEL
LIN {X 0,Y 153.104,Z 460.183,A -85,B 0,C 180,E1 -23870.137,E2 -23870.137} C_VEL
LIN {X 0,Y 155.159,Z 457.808,A -85,B 0,C 180,E1 -23872.644,E2 -23872.644} C_VEL
LIN {X 0,Y 158.862,Z 452.983,A -85,B 0,C 180,E1 -23876.256,E2 -23876.256} C_VEL
LIN {X 0,Y 162.437,Z 447.807,A -85,B 0,C 180,E1 -23879.126,E2 -23879.126} C_VEL
LIN {X 0,Y 165.658,Z 442.765,A -85,B 0,C 180,E1 -23881.312,E2 -23881.312} C_VEL
LIN {X 0,Y 169.017,Z 436.733,A -85,B 0,C 180,E1 -23883.432,E2 -23883.432} C_VEL
LIN {X 0,Y 172.355,Z 430.246,A -85,B 0,C 180,E1 -23885.229,E2 -23885.229} C_VEL
LIN {X 0,Y 175.683,Z 422.808,A -85,B 0,C 180,E1 -23886.874,E2 -23886.874} C_VEL
LIN {X 0,Y 178.762,Z 414.836,A -85,B 0,C 180,E1 -23888.258,E2 -23888.258} C_VEL
LIN {X 0,Y 181.478,Z 406.6,A -85,B 0,C 180,E1 -23889.356,E2 -23889.356} C_VEL
LIN {X 0,Y 183.744,Z 398.243,A -85,B 0,C 180,E1 -23890.199,E2 -23890.199} C_VEL
LIN {X 0,Y 185.634,Z 388.555,A -85,B 0,C 180,E1 -23890.941,E2 -23890.941} C_VEL
LIN {X 0,Y 187.002,Z 377.9,A -85,B 0,C 180,E1 -23891.468,E2 -23891.468} C_VEL
LIN {X 0,Y 187.488,Z 369.761,A -85,B 0,C 180,E1 -23891.799,E2 -23891.799} C_VEL
LIN {X 0,Y 186.768,Z 362.48,A -85,B 0,C 180,E1 -23892.48,E2 -23892.48} C_VEL
LIN {X 0,Y 181.888,Z 350.53,A -85,B 0,C 180,E1 -23895.062,E2 -23895.062} C_VEL
LIN {X 0,Y 178.062,Z 342.602,A -85,B 0,C 180,E1 -23897.203,E2 -23897.203} C_VEL
LIN {X 0,Y 173.805,Z 334.766,A -85,B 0,C 180,E1 -23899.77,E2 -23899.77} C_VEL
LIN {X 0,Y 170.743,Z 329.555,A -85,B 0,C 180,E1 -23901.781,E2 -23901.781} C_VEL
LIN {X 0,Y 167.98,Z 324.866,A -85,B 0,C 180,E1 -23903.809,E2 -23903.809} C_VEL
LIN {X 0,Y 164.553,Z 319.527,A -85,B 0,C 180,E1 -23906.587,E2 -23906.587} C_VEL
LIN {X 0,Y 160.651,Z 313.956,A -85,B 0,C 180,E1 -23910.241,E2 -23910.241} C_VEL
LIN {X 0,Y 160.106,Z 313.164,A -85,B 0,C 180,E1 -23910.813,E2 -23910.813} C_VEL
LIN {X 0,Y 157.484,Z 311.202,A -85,B 0,C 180,E1 -23913.606,E2 -23913.606} C_VEL
LIN {X 0,Y 155.932,Z 308.318,A -85,B 0,C 180,E1 -23915.807,E2 -23915.807} C_VEL
LIN {X 0,Y 155.588,Z 307.591,A -85,B 0,C 180,E1 -23916.358,E2 -23916.358} C_VEL
LIN {X 0,Y 152.001,Z 305.307,A -85,B 0,C 180,E1 -23922.849,E2 -23922.849} C_VEL
LIN {X 0,Y 150.709,Z 302.226,A -85,B 0,C 180,E1 -23928.522,E2 -23928.522} C_VEL
LIN {X 0,Y 150.655,Z 301.51,A -85,B 0,C 180,E1 -23929.917,E2 -23929.917} C_VEL
LIN {X 0,Y 150.662,Z 301.615,A -85,B 0,C 180,E1 -23934.303,E2 -23934.303} C_VEL
LIN {X 0,Y 151.865,Z 303.688,A -85,B 0,C 180,E1 -23939.991,E2 -23939.991} C_VEL
LIN {X 0,Y 153.468,Z 306.265,A -85,B 0,C 180,E1 -23943.93,E2 -23943.93} C_VEL
LIN {X 0,Y 156.118,Z 307.802,A -85,B 0,C 180,E1 -23948.017,E2 -23948.017} C_VEL
LIN {X 0,Y 157.563,Z 310.787,A -85,B 0,C 180,E1 -23950.09,E2 -23950.09} C_VEL
LIN {X 0,Y 159.939,Z 312.975,A -85,B 0,C 180,E1 -23952.683,E2 -23952.683} C_VEL
LIN {X 0,Y 160.524,Z 313.457,A -85,B 0,C 180,E1 -23953.26,E2 -23953.26} C_VEL
LIN {X 0,Y 162.515,Z 316.699,A -85,B 0,C 180,E1 -23955.271,E2 -23955.271} C_VEL
LIN {X 0,Y 164.745,Z 318.876,A -85,B 0,C 180,E1 -23957.156,E2 -23957.156} C_VEL
LIN {X 0,Y 167.304,Z 322.536,A -85,B 0,C 180,E1 -23959.224,E2 -23959.224} C_VEL
LIN {X 0,Y 168.616,Z 324.113,A -85,B 0,C 180,E1 -23960.183,E2 -23960.183} C_VEL
LIN {X 0,Y 172.098,Z 329.008,A -85,B 0,C 180,E1 -23962.586,E2 -23962.586} C_VEL
LIN {X 0,Y 175.241,Z 333.502,A -85,B 0,C 180,E1 -23964.519,E2 -23964.519} C_VEL
LIN {X 0,Y 179.709,Z 340.278,A -85,B 0,C 180,E1 -23967.032,E2 -23967.032} C_VEL
LIN {X 0,Y 185.822,Z 350.771,A -85,B 0,C 180,E1 -23970.144,E2 -23970.144} C_VEL
LIN {X 0,Y 188.456,Z 355.805,A -85,B 0,C 180,E1 -23971.395,E2 -23971.395} C_VEL
LIN {X 0,Y 187.113,Z 372.787,A -85,B 0,C 180,E1 -23972.083,E2 -23972.083} C_VEL
LIN {X 0,Y 185.244,Z 384.362,A -85,B 0,C 180,E1 -23972.931,E2 -23972.931} C_VEL
LIN {X 0,Y 183.133,Z 393.619,A -85,B 0,C 180,E1 -23973.913,E2 -23973.913} C_VEL
LIN {X 0,Y 180.531,Z 402.521,A -85,B 0,C 180,E1 -23975.163,E2 -23975.163} C_VEL
LIN {X 0,Y 177.703,Z 410.267,A -85,B 0,C 180,E1 -23976.53,E2 -23976.53} C_VEL
LIN {X 0,Y 174.528,Z 417.88,A -85,B 0,C 180,E1 -23978.258,E2 -23978.258} C_VEL
LIN {X 0,Y 170.814,Z 425.463,A -85,B 0,C 180,E1 -23980.434,E2 -23980.434} C_VEL
LIN {X 0,Y 166.341,Z 433.113,A -85,B 0,C 180,E1 -23983.303,E2 -23983.303} C_VEL
LIN {X 0,Y 162.457,Z 438.791,A -85,B 0,C 180,E1 -23986.198,E2 -23986.198} C_VEL
LIN {X 0,Y 159.614,Z 442.551,A -85,B 0,C 180,E1 -23988.665,E2 -23988.665} C_VEL
LIN {X 0,Y 157.064,Z 445.592,A -85,B 0,C 180,E1 -23991.212,E2 -23991.212} C_VEL
LIN {X 0,Y 154.838,Z 447.947,A -85,B 0,C 180,E1 -23993.839,E2 -23993.839} C_VEL
LIN {X 0,Y 152.921,Z 449.635,A -85,B 0,C 180,E1 -23996.53,E2 -23996.53} C_VEL
LIN {X 0,Y 151.269,Z 450.746,A -85,B 0,C 180,E1 -23999.266,E2 -23999.266} C_VEL
LIN {X 0,Y 149.462,Z 451.451,A -85,B 0,C 180,E1 -24003.282,E2 -24003.282} C_VEL
LIN {X 0,Y 148.194,Z 450.927,A -85,B 0,C 180,E1 -24007.704,E2 -24007.704} C_VEL
LIN {X 0,Y 147.638,Z 448.989,A -85,B 0,C 180,E1 -24012.151,E2 -24012.151} C_VEL
LIN {X 0,Y 147.71,Z 446.029,A -85,B 0,C 180,E1 -24016.238,E2 -24016.238} C_VEL
LIN {X 0,Y 148.043,Z 443.232,A -85,B 0,C 180,E1 -24019.054,E2 -24019.054} C_VEL
LIN {X 0,Y 148.826,Z 438.812,A -85,B 0,C 180,E1 -24022.52,E2 -24022.52} C_VEL
LIN {X 0,Y 149.848,Z 433.184,A -85,B 0,C 180,E1 -24025.966,E2 -24025.966} C_VEL
LIN {X 0,Y 151.162,Z 426.186,A -85,B 0,C 180,E1 -24029.335,E2 -24029.335} C_VEL
LIN {X 0,Y 152.769,Z 418.112,A -85,B 0,C 180,E1 -24032.308,E2 -24032.308} C_VEL
LIN {X 0,Y 154.298,Z 410.377,A -85,B 0,C 180,E1 -24034.572,E2 -24034.572} C_VEL
LIN {X 0,Y 155.652,Z 402.723,A -85,B 0,C 180,E1 -24036.385,E2 -24036.385} C_VEL
LIN {X 0,Y 156.987,Z 393.888,A -85,B 0,C 180,E1 -24038.043,E2 -24038.043} C_VEL
LIN {X 0,Y 157.956,Z 385.41,A -85,B 0,C 180,E1 -24039.282,E2 -24039.282} C_VEL
LIN {X 0,Y 158.909,Z 375.557,A -85,B 0,C 180,E1 -24040.326,E2 -24040.326} C_VEL
LIN {X 0,Y 159.564,Z 364.526,A -85,B 0,C 180,E1 -24041.081,E2 -24041.081} C_VEL
LIN {X 0,Y 160.962,Z 326.42,A -85,B 0,C 180,E1 -24042.743,E2 -24042.743} C_VEL
LIN {X 0,Y 157.088,Z 316.336,A -85,B 0,C 180,E1 -24043.866,E2 -24043.866} C_VEL
LIN {X 0,Y 150.461,Z 302.209,A -85,B 0,C 180,E1 -24045.768,E2 -24045.768} C_VEL
LIN {X 0,Y 150.345,Z 301.568,A -85,B 0,C 180,E1 -24045.879,E2 -24045.879} C_VEL
LIN {X 0,Y 150.324,Z 301.572,A -85,B 0,C 180,E1 -24050.794,E2 -24050.794} C_VEL
LIN {X 0,Y 150.215,Z 301.587,A -85,B 0,C 180,E1 -24057.282,E2 -24057.282} C_VEL
LIN {X 0,Y 150.182,Z 301.579,A -85,B 0,C 180,E1 -24062.632,E2 -24062.632} C_VEL
LIN {X 0,Y 150.148,Z 301.59,A -85,B 0,C 180,E1 -24067.481,E2 -24067.481} C_VEL
LIN {X 0,Y 150.114,Z 301.598,A -85,B 0,C 180,E1 -24071.504,E2 -24071.504} C_VEL
LIN {X 0,Y 150.108,Z 301.595,A -85,B 0,C 180,E1 -24075.403,E2 -24075.403} C_VEL
LIN {X 0,Y 150.125,Z 301.595,A -85,B 0,C 180,E1 -24079.063,E2 -24079.063} C_VEL
LIN {X 0,Y 150.165,Z 301.591,A -85,B 0,C 180,E1 -24082.716,E2 -24082.716} C_VEL
LIN {X 0,Y 150.196,Z 301.583,A -85,B 0,C 180,E1 -24087.381,E2 -24087.381} C_VEL
